KUKA KRL program: EPS_2_251806_MH45A_A_20260212042240.src

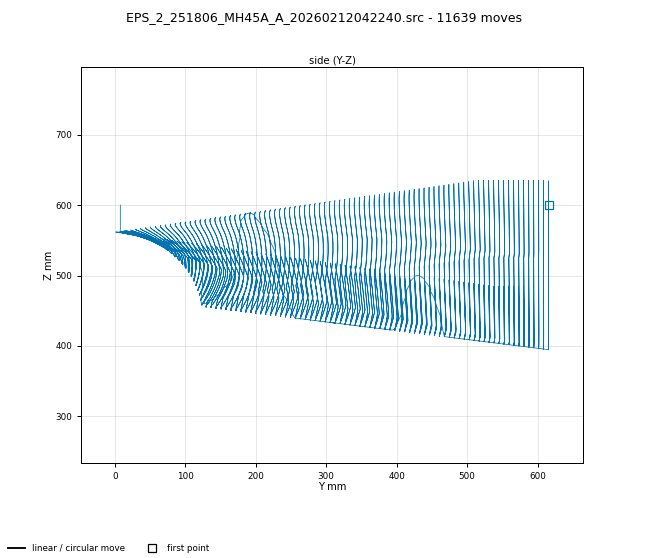
[picture p0: tool path of EPS_2_251806_MH45A_A_20260212042240.src, 11639 of 11641 moves have a stored position in this frame; points joined in program order, loops and branches not executed]
&ACCESS RVP
&REL 4
&COMMENT QRS 19112012
&PARAM EDITMASK = *
DEF PART()
EXT BAS (BAS_COMMAND :IN,REAL :IN )
INT I
BAS (#INITMOV,0 )

;KUKA QRS Post kuka4.cps  Date:22-06-2017 !

File_ID=3017

QRS_PRE_INIT()

;Init var - Until changes are made in qrs_pre_init
Outlet_Square_prg=0
Inlet_1_Square_prg=0
Inlet_2_Square_prg=0
Inlet_3_Square_prg=0
Inlet_4_Square_prg=0
Inlet_5_Square_prg=0

Outlet_1={X 0.000, Y 515.340, Z 534.500, B 0.000, E1 0.000 }
Inlet_1={X 0.000, Y 533.470, Z 284.500, B 0.000, E1 180.000 }
Outlet_1_type=201
Inlet_1_type=201
;QRS#1=Sidecore dimensions
;QRS#2=200-8" PVC SDR 35
;QRS#3=200-8" PVC SDR 35
;QRS#4=
;QRS#5=
;QRS#6=
;QRS#7=
;QRS#8=
;QRS#9=12-08 PSX
;QRS#10=12-08 PSX
;QRS#11=
;QRS#12=
;QRS#13=
;QRS#14=
;QRS#15=
;QRS#16=1220x127x914 3'
;QRS#17=EPS Height
;QRS#18=635
;QRS#19=*
;QRS#20= UPDATED VERSION 22-06-2017
;QRS#21=*
Outlet_Square=0100
Inlet_1_Square=0100
Inlet_2_Square=0
Inlet_3_Square=0
Inlet_4_Square=0
Inlet_5_Square=0
Mill_Square=1
Outlet_Square_Prg=204
Inlet_1_Square_prg=204

QRS_INIT()

$ADVANCE=5

; T1
PTP {E1 173.608,E2 173.608}
PTP {X 0,Y 615.507,A -85,B 0,C 180,E1 173.608,E2 173.608,E3 0,E4 0,E5 0,E6 0}
QRS_SPEED_INIT()
LIN {X 0,Y 615.507,Z 600,A -85,B 0,C 180,E1 173.608,E2 173.608,E3 0,E4 0,E5 0,E6 0} C_VEL
LIN {X 0,Y 615.507,Z 404.876,A -85,B 0,C 180,E1 173.608,E2 173.608} C_VEL
LIN {X 0,Y 615.507,Z 396.699,A -85,B 0,C 180,E1 173.608,E2 173.608} C_VEL
LIN {X 0,Y 615.491,Z 394.699,A -85,B 0,C 180,E1 173.422,E2 173.422} C_VEL
LIN {X 0,Y 615.482,Z 394.699,A -85,B 0,C 180,E1 170.801,E2 170.801} C_VEL
LIN {X 0,Y 615.49,Z 394.7,A -85,B 0,C 180,E1 168.139,E2 168.139} C_VEL
LIN {X 0,Y 615.496,Z 394.696,A -85,B 0,C 180,E1 165.451,E2 165.451} C_VEL
LIN {X 0,Y 615.497,Z 394.697,A -85,B 0,C 180,E1 162.73,E2 162.73} C_VEL
LIN {X 0,Y 615.486,Z 394.7,A -85,B 0,C 180,E1 159.967,E2 159.967} C_VEL
LIN {X 0,Y 615.477,Z 394.699,A -85,B 0,C 180,E1 157.155,E2 157.155} C_VEL
LIN {X 0,Y 615.496,Z 394.7,A -85,B 0,C 180,E1 154.43,E2 154.43} C_VEL
LIN {X 0,Y 615.497,Z 394.697,A -85,B 0,C 180,E1 151.549,E2 151.549} C_VEL
LIN {X 0,Y 615.491,Z 394.697,A -85,B 0,C 180,E1 148.914,E2 148.914} C_VEL
LIN {X 0,Y 615.485,Z 394.698,A -85,B 0,C 180,E1 146.467,E2 146.467} C_VEL
LIN {X 0,Y 615.49,Z 394.697,A -85,B 0,C 180,E1 143.575,E2 143.575} C_VEL
LIN {X 0,Y 615.481,Z 394.7,A -85,B 0,C 180,E1 140.939,E2 140.939} C_VEL
LIN {X 0,Y 615.495,Z 394.7,A -85,B 0,C 180,E1 138.527,E2 138.527} C_VEL
LIN {X 0,Y 615.494,Z 394.696,A -85,B 0,C 180,E1 135.851,E2 135.851} C_VEL
LIN {X 0,Y 615.487,Z 394.699,A -85,B 0,C 180,E1 133.047,E2 133.047} C_VEL
LIN {X 0,Y 615.479,Z 394.699,A -85,B 0,C 180,E1 130.607,E2 130.607} C_VEL
LIN {X 0,Y 615.488,Z 394.702,A -85,B 0,C 180,E1 128.012,E2 128.012} C_VEL
LIN {X 0,Y 615.486,Z 394.699,A -85,B 0,C 180,E1 125.616,E2 125.616} C_VEL
LIN {X 0,Y 615.479,Z 394.699,A -85,B 0,C 180,E1 123.237,E2 123.237} C_VEL
LIN {X 0,Y 615.493,Z 394.697,A -85,B 0,C 180,E1 120.92,E2 120.92} C_VEL
LIN {X 0,Y 615.497,Z 394.7,A -85,B 0,C 180,E1 118.451,E2 118.451} C_VEL
LIN {X 0,Y 615.492,Z 394.697,A -85,B 0,C 180,E1 115.569,E2 115.569} C_VEL
LIN {X 0,Y 615.49,Z 394.697,A -85,B 0,C 180,E1 112.845,E2 112.845} C_VEL
LIN {X 0,Y 615.487,Z 394.702,A -85,B 0,C 180,E1 110.033,E2 110.033} C_VEL
LIN {X 0,Y 615.477,Z 394.699,A -85,B 0,C 180,E1 107.271,E2 107.271} C_VEL
LIN {X 0,Y 615.49,Z 394.7,A -85,B 0,C 180,E1 104.549,E2 104.549} C_VEL
LIN {X 0,Y 615.494,Z 394.696,A -85,B 0,C 180,E1 101.861,E2 101.861} C_VEL
LIN {X 0,Y 615.487,Z 394.736,A -85,B 0,C 180,E1 101.235,E2 101.235} C_VEL
LIN {X 0,Y 615.485,Z 406.659,A -85,B 0,C 180,E1 100.84,E2 100.84} C_VEL
LIN {X 0,Y 615.494,Z 419.193,A -85,B 0,C 180,E1 100.277,E2 100.277} C_VEL
LIN {X 0,Y 615.493,Z 430.575,A -85,B 0,C 180,E1 99.613,E2 99.613} C_VEL
LIN {X 0,Y 615.498,Z 440.821,A -85,B 0,C 180,E1 98.867,E2 98.867} C_VEL
LIN {X 0,Y 615.499,Z 450.033,A -85,B 0,C 180,E1 98.041,E2 98.041} C_VEL
LIN {X 0,Y 615.499,Z 458.891,A -85,B 0,C 180,E1 97.057,E2 97.057} C_VEL
LIN {X 0,Y 615.497,Z 466.123,A -85,B 0,C 180,E1 96.063,E2 96.063} C_VEL
LIN {X 0,Y 615.497,Z 470.957,A -85,B 0,C 180,E1 95.241,E2 95.241} C_VEL
LIN {X 0,Y 615.494,Z 475.657,A -85,B 0,C 180,E1 94.256,E2 94.256} C_VEL
LIN {X 0,Y 615.494,Z 479.254,A -85,B 0,C 180,E1 93.273,E2 93.273} C_VEL
LIN {X 0,Y 615.496,Z 481.115,A -85,B 0,C 180,E1 92.618,E2 92.618} C_VEL
LIN {X 0,Y 615.499,Z 482.533,A -85,B 0,C 180,E1 91.963,E2 91.963} C_VEL
LIN {X 0,Y 615.496,Z 484.141,A -85,B 0,C 180,E1 90.654,E2 90.654} C_VEL
LIN {X 0,Y 615.495,Z 484.384,A -85,B 0,C 180,E1 90,E2 90} C_VEL
LIN {X 0,Y 615.495,Z 484.206,A -85,B 0,C 180,E1 89.346,E2 89.346} C_VEL
LIN {X 0,Y 615.499,Z 482.682,A -85,B 0,C 180,E1 88.037,E2 88.037} C_VEL
LIN {X 0,Y 615.498,Z 481.341,A -85,B 0,C 180,E1 87.382,E2 87.382} C_VEL
LIN {X 0,Y 615.496,Z 478.494,A -85,B 0,C 180,E1 86.399,E2 86.399} C_VEL
LIN {X 0,Y 615.499,Z 474.634,A -85,B 0,C 180,E1 85.416,E2 85.416} C_VEL
LIN {X 0,Y 615.498,Z 469.652,A -85,B 0,C 180,E1 84.43,E2 84.43} C_VEL
LIN {X 0,Y 615.496,Z 463.208,A -85,B 0,C 180,E1 83.418,E2 83.418} C_VEL
LIN {X 0,Y 615.497,Z 455.537,A -85,B 0,C 180,E1 82.455,E2 82.455} C_VEL
LIN {X 0,Y 615.498,Z 445.759,A -85,B 0,C 180,E1 81.464,E2 81.464} C_VEL
LIN {X 0,Y 615.498,Z 435.493,A -85,B 0,C 180,E1 80.636,E2 80.636} C_VEL
LIN {X 0,Y 615.492,Z 423.93,A -85,B 0,C 180,E1 79.889,E2 79.889} C_VEL
LIN {X 0,Y 615.485,Z 412.104,A -85,B 0,C 180,E1 79.294,E2 79.294} C_VEL
LIN {X 0,Y 615.486,Z 399.16,A -85,B 0,C 180,E1 78.807,E2 78.807} C_VEL
LIN {X 0,Y 615.485,Z 394.699,A -85,B 0,C 180,E1 78.661,E2 78.661} C_VEL
LIN {X 0,Y 615.499,Z 394.696,A -85,B 0,C 180,E1 76.064,E2 76.064} C_VEL
LIN {X 0,Y 615.481,Z 394.699,A -85,B 0,C 180,E1 73.413,E2 73.413} C_VEL
LIN {X 0,Y 615.483,Z 394.699,A -85,B 0,C 180,E1 70.662,E2 70.662} C_VEL
LIN {X 0,Y 615.495,Z 394.7,A -85,B 0,C 180,E1 67.864,E2 67.864} C_VEL
LIN {X 0,Y 615.489,Z 394.697,A -85,B 0,C 180,E1 65.008,E2 65.008} C_VEL
LIN {X 0,Y 615.488,Z 394.698,A -85,B 0,C 180,E1 62.823,E2 62.823} C_VEL
LIN {X 0,Y 615.499,Z 394.697,A -85,B 0,C 180,E1 60.204,E2 60.204} C_VEL
LIN {X 0,Y 615.481,Z 394.699,A -85,B 0,C 180,E1 57.542,E2 57.542} C_VEL
LIN {X 0,Y 615.499,Z 394.699,A -85,B 0,C 180,E1 55.186,E2 55.186} C_VEL
LIN {X 0,Y 615.488,Z 394.699,A -85,B 0,C 180,E1 52.758,E2 52.758} C_VEL
LIN {X 0,Y 615.497,Z 394.699,A -85,B 0,C 180,E1 49.91,E2 49.91} C_VEL
LIN {X 0,Y 615.496,Z 394.7,A -85,B 0,C 180,E1 47.648,E2 47.648} C_VEL
LIN {X 0,Y 615.481,Z 394.699,A -85,B 0,C 180,E1 44.931,E2 44.931} C_VEL
LIN {X 0,Y 615.487,Z 394.698,A -85,B 0,C 180,E1 42.08,E2 42.08} C_VEL
LIN {X 0,Y 615.477,Z 394.699,A -85,B 0,C 180,E1 39.751,E2 39.751} C_VEL
LIN {X 0,Y 615.486,Z 394.7,A -85,B 0,C 180,E1 36.936,E2 36.936} C_VEL
LIN {X 0,Y 615.494,Z 394.7,A -85,B 0,C 180,E1 34.022,E2 34.022} C_VEL
LIN {X 0,Y 615.489,Z 394.7,A -85,B 0,C 180,E1 31.686,E2 31.686} C_VEL
LIN {X 0,Y 615.492,Z 394.697,A -85,B 0,C 180,E1 29.406,E2 29.406} C_VEL
LIN {X 0,Y 615.495,Z 394.7,A -85,B 0,C 180,E1 26.444,E2 26.444} C_VEL
LIN {X 0,Y 615.486,Z 394.699,A -85,B 0,C 180,E1 23.557,E2 23.557} C_VEL
LIN {X 0,Y 615.484,Z 394.698,A -85,B 0,C 180,E1 20.731,E2 20.731} C_VEL
LIN {X 0,Y 615.49,Z 394.701,A -85,B 0,C 180,E1 17.957,E2 17.957} C_VEL
LIN {X 0,Y 615.486,Z 394.698,A -85,B 0,C 180,E1 15.226,E2 15.226} C_VEL
LIN {X 0,Y 615.494,Z 394.698,A -85,B 0,C 180,E1 12.53,E2 12.53} C_VEL
LIN {X 0,Y 615.481,Z 394.7,A -85,B 0,C 180,E1 9.862,E2 9.862} C_VEL
LIN {X 0,Y 615.484,Z 394.7,A -85,B 0,C 180,E1 7.216,E2 7.216} C_VEL
LIN {X 0,Y 615.489,Z 394.697,A -85,B 0,C 180,E1 4.585,E2 4.585} C_VEL
LIN {X 0,Y 615.484,Z 394.7,A -85,B 0,C 180,E1 1.963,E2 1.963} C_VEL
LIN {X 0,Y 615.485,Z 394.698,A -85,B 0,C 180,E1 -0.654,E2 -0.654} C_VEL
LIN {X 0,Y 615.498,Z 394.698,A -85,B 0,C 180,E1 -3.273,E2 -3.273} C_VEL
LIN {X 0,Y 615.483,Z 394.698,A -85,B 0,C 180,E1 -5.899,E2 -5.899} C_VEL
LIN {X 0,Y 615.486,Z 394.701,A -85,B 0,C 180,E1 -8.537,E2 -8.537} C_VEL
LIN {X 0,Y 615.486,Z 394.698,A -85,B 0,C 180,E1 -11.193,E2 -11.193} C_VEL
LIN {X 0,Y 615.487,Z 394.699,A -85,B 0,C 180,E1 -13.932,E2 -13.932} C_VEL
LIN {X 0,Y 615.487,Z 394.698,A -85,B 0,C 180,E1 -16.587,E2 -16.587} C_VEL
LIN {X 0,Y 615.493,Z 394.697,A -85,B 0,C 180,E1 -19.338,E2 -19.338} C_VEL
LIN {X 0,Y 615.494,Z 394.699,A -85,B 0,C 180,E1 -22.347,E2 -22.347} C_VEL
LIN {X 0,Y 615.477,Z 394.7,A -85,B 0,C 180,E1 -24.992,E2 -24.992} C_VEL
LIN {X 0,Y 615.485,Z 394.698,A -85,B 0,C 180,E1 -27.177,E2 -27.177} C_VEL
LIN {X 0,Y 615.481,Z 394.701,A -85,B 0,C 180,E1 -29.793,E2 -29.793} C_VEL
LIN {X 0,Y 615.487,Z 394.698,A -85,B 0,C 180,E1 -32.458,E2 -32.458} C_VEL
LIN {X 0,Y 615.49,Z 394.7,A -85,B 0,C 180,E1 -34.815,E2 -34.815} C_VEL
LIN {X 0,Y 615.493,Z 394.698,A -85,B 0,C 180,E1 -37.242,E2 -37.242} C_VEL
LIN {X 0,Y 615.491,Z 394.7,A -85,B 0,C 180,E1 -40.089,E2 -40.089} C_VEL
LIN {X 0,Y 615.498,Z 394.7,A -85,B 0,C 180,E1 -42.352,E2 -42.352} C_VEL
LIN {X 0,Y 615.485,Z 394.698,A -85,B 0,C 180,E1 -45.069,E2 -45.069} C_VEL
LIN {X 0,Y 615.481,Z 394.7,A -85,B 0,C 180,E1 -47.921,E2 -47.921} C_VEL
LIN {X 0,Y 615.494,Z 394.695,A -85,B 0,C 180,E1 -50.25,E2 -50.25} C_VEL
LIN {X 0,Y 615.495,Z 394.699,A -85,B 0,C 180,E1 -53.063,E2 -53.063} C_VEL
LIN {X 0,Y 615.481,Z 394.823,A -85,B 0,C 180,E1 -54.534,E2 -54.534} C_VEL
LIN {X 0,Y 615.489,Z 408.627,A -85,B 0,C 180,E1 -57.154,E2 -57.154} C_VEL
LIN {X 0,Y 615.476,Z 422.322,A -85,B 0,C 180,E1 -59.839,E2 -59.839} C_VEL
LIN {X 0,Y 615.481,Z 436.017,A -85,B 0,C 180,E1 -62.454,E2 -62.454} C_VEL
LIN {X 0,Y 615.497,Z 449.706,A -85,B 0,C 180,E1 -65.009,E2 -65.009} C_VEL
LIN {X 0,Y 615.487,Z 465.338,A -85,B 0,C 180,E1 -67.864,E2 -67.864} C_VEL
LIN {X 0,Y 615.492,Z 480.954,A -85,B 0,C 180,E1 -70.662,E2 -70.662} C_VEL
LIN {X 0,Y 615.492,Z 496.556,A -85,B 0,C 180,E1 -73.413,E2 -73.413} C_VEL
LIN {X 0,Y 615.498,Z 512.142,A -85,B 0,C 180,E1 -76.126,E2 -76.126} C_VEL
LIN {X 0,Y 615.482,Z 524.941,A -85,B 0,C 180,E1 -78.327,E2 -78.327} C_VEL
LIN {X 0,Y 615.477,Z 538.242,A -85,B 0,C 180,E1 -78.557,E2 -78.557} C_VEL
LIN {X 0,Y 615.489,Z 551.335,A -85,B 0,C 180,E1 -78.922,E2 -78.922} C_VEL
LIN {X 0,Y 615.48,Z 563.13,A -85,B 0,C 180,E1 -79.383,E2 -79.383} C_VEL
LIN {X 0,Y 615.486,Z 574.575,A -85,B 0,C 180,E1 -79.972,E2 -79.972} C_VEL
LIN {X 0,Y 615.499,Z 586.021,A -85,B 0,C 180,E1 -80.719,E2 -80.719} C_VEL
LIN {X 0,Y 615.498,Z 595.257,A -85,B 0,C 180,E1 -81.464,E2 -81.464} C_VEL
LIN {X 0,Y 615.499,Z 603.654,A -85,B 0,C 180,E1 -82.29,E2 -82.29} C_VEL
LIN {X 0,Y 615.497,Z 611.69,A -85,B 0,C 180,E1 -83.259,E2 -83.259} C_VEL
LIN {X 0,Y 615.498,Z 617.423,A -85,B 0,C 180,E1 -84.102,E2 -84.102} C_VEL
LIN {X 0,Y 615.497,Z 622.872,A -85,B 0,C 180,E1 -85.087,E2 -85.087} C_VEL
LIN {X 0,Y 615.496,Z 627.141,A -85,B 0,C 180,E1 -86.072,E2 -86.072} C_VEL
LIN {X 0,Y 615.495,Z 629.399,A -85,B 0,C 180,E1 -86.727,E2 -86.727} C_VEL
LIN {X 0,Y 615.497,Z 631.233,A -85,B 0,C 180,E1 -87.382,E2 -87.382} C_VEL
LIN {X 0,Y 615.497,Z 632.608,A -85,B 0,C 180,E1 -88.037,E2 -88.037} C_VEL
LIN {X 0,Y 615.496,Z 634.174,A -85,B 0,C 180,E1 -89.346,E2 -89.346} C_VEL
LIN {X 0,Y 615.494,Z 634.389,A -85,B 0,C 180,E1 -90,E2 -90} C_VEL
LIN {X 0,Y 615.496,Z 633.58,A -85,B 0,C 180,E1 -91.309,E2 -91.309} C_VEL
LIN {X 0,Y 615.497,Z 632.608,A -85,B 0,C 180,E1 -91.963,E2 -91.963} C_VEL
LIN {X 0,Y 615.497,Z 631.233,A -85,B 0,C 180,E1 -92.618,E2 -92.618} C_VEL
LIN {X 0,Y 615.496,Z 628.349,A -85,B 0,C 180,E1 -93.601,E2 -93.601} C_VEL
LIN {X 0,Y 615.498,Z 624.441,A -85,B 0,C 180,E1 -94.585,E2 -94.585} C_VEL
LIN {X 0,Y 615.499,Z 619.404,A -85,B 0,C 180,E1 -95.57,E2 -95.57} C_VEL
LIN {X 0,Y 615.497,Z 612.869,A -85,B 0,C 180,E1 -96.583,E2 -96.583} C_VEL
LIN {X 0,Y 615.497,Z 605.132,A -85,B 0,C 180,E1 -97.545,E2 -97.545} C_VEL
LIN {X 0,Y 615.498,Z 597.044,A -85,B 0,C 180,E1 -98.371,E2 -98.371} C_VEL
LIN {X 0,Y 615.499,Z 587.166,A -85,B 0,C 180,E1 -99.199,E2 -99.199} C_VEL
LIN {X 0,Y 615.488,Z 575.98,A -85,B 0,C 180,E1 -99.945,E2 -99.945} C_VEL
LIN {X 0,Y 615.478,Z 565.022,A -85,B 0,C 180,E1 -100.527,E2 -100.527} C_VEL
LIN {X 0,Y 615.489,Z 552.502,A -85,B 0,C 180,E1 -101.04,E2 -101.04} C_VEL
LIN {X 0,Y 615.477,Z 540.062,A -85,B 0,C 180,E1 -101.402,E2 -101.402} C_VEL
LIN {X 0,Y 615.481,Z 526.459,A -85,B 0,C 180,E1 -101.652,E2 -101.652} C_VEL
LIN {X 0,Y 615.483,Z 524.798,A -85,B 0,C 180,E1 -101.694,E2 -101.694} C_VEL
LIN {X 0,Y 615.48,Z 510.016,A -85,B 0,C 180,E1 -104.243,E2 -104.243} C_VEL
LIN {X 0,Y 615.494,Z 494.604,A -85,B 0,C 180,E1 -106.928,E2 -106.928} C_VEL
LIN {X 0,Y 615.495,Z 479.001,A -85,B 0,C 180,E1 -109.685,E2 -109.685} C_VEL
LIN {X 0,Y 615.494,Z 462.801,A -85,B 0,C 180,E1 -112.595,E2 -112.595} C_VEL
LIN {X 0,Y 615.485,Z 448.151,A -85,B 0,C 180,E1 -115.279,E2 -115.279} C_VEL
LIN {X 0,Y 615.493,Z 434.06,A -85,B 0,C 180,E1 -117.915,E2 -117.915} C_VEL
LIN {X 0,Y 615.478,Z 420.365,A -85,B 0,C 180,E1 -120.54,E2 -120.54} C_VEL
LIN {X 0,Y 615.491,Z 406.663,A -85,B 0,C 180,E1 -123.236,E2 -123.236} C_VEL
LIN {X 0,Y 615.482,Z 394.698,A -85,B 0,C 180,E1 -125.516,E2 -125.516} C_VEL
LIN {X 0,Y 615.498,Z 394.699,A -85,B 0,C 180,E1 -128.068,E2 -128.068} C_VEL
LIN {X 0,Y 615.491,Z 394.697,A -85,B 0,C 180,E1 -130.606,E2 -130.606} C_VEL
LIN {X 0,Y 615.491,Z 394.698,A -85,B 0,C 180,E1 -133.245,E2 -133.245} C_VEL
LIN {X 0,Y 615.484,Z 394.698,A -85,B 0,C 180,E1 -136.003,E2 -136.003} C_VEL
LIN {X 0,Y 615.485,Z 394.7,A -85,B 0,C 180,E1 -138.526,E2 -138.526} C_VEL
LIN {X 0,Y 615.484,Z 394.7,A -85,B 0,C 180,E1 -141.095,E2 -141.095} C_VEL
LIN {X 0,Y 615.489,Z 394.697,A -85,B 0,C 180,E1 -143.575,E2 -143.575} C_VEL
LIN {X 0,Y 615.494,Z 394.697,A -85,B 0,C 180,E1 -146.465,E2 -146.465} C_VEL
LIN {X 0,Y 615.49,Z 394.698,A -85,B 0,C 180,E1 -149.08,E2 -149.08} C_VEL
LIN {X 0,Y 615.498,Z 394.699,A -85,B 0,C 180,E1 -151.549,E2 -151.549} C_VEL
LIN {X 0,Y 615.484,Z 394.7,A -85,B 0,C 180,E1 -154.433,E2 -154.433} C_VEL
LIN {X 0,Y 615.48,Z 394.699,A -85,B 0,C 180,E1 -157.155,E2 -157.155} C_VEL
LIN {X 0,Y 615.491,Z 394.701,A -85,B 0,C 180,E1 -159.967,E2 -159.967} C_VEL
LIN {X 0,Y 615.495,Z 394.696,A -85,B 0,C 180,E1 -162.73,E2 -162.73} C_VEL
LIN {X 0,Y 615.497,Z 394.697,A -85,B 0,C 180,E1 -165.451,E2 -165.451} C_VEL
LIN {X 0,Y 615.484,Z 394.699,A -85,B 0,C 180,E1 -168.139,E2 -168.139} C_VEL
LIN {X 0,Y 615.479,Z 394.7,A -85,B 0,C 180,E1 -170.801,E2 -170.801} C_VEL
LIN {X 0,Y 615.492,Z 394.697,A -85,B 0,C 180,E1 -173.443,E2 -173.443} C_VEL
LIN {X 0,Y 615.49,Z 394.698,A -85,B 0,C 180,E1 -176.072,E2 -176.072} C_VEL
LIN {X 0,Y 615.495,Z 394.696,A -85,B 0,C 180,E1 -178.691,E2 -178.691} C_VEL
LIN {X 0,Y 615.496,Z 394.698,A -85,B 0,C 180,E1 -181.309,E2 -181.309} C_VEL
LIN {X 0,Y 615.48,Z 394.699,A -85,B 0,C 180,E1 -183.929,E2 -183.929} C_VEL
LIN {X 0,Y 615.491,Z 394.699,A -85,B 0,C 180,E1 -186.578,E2 -186.578} C_VEL
LIN {X 0,Y 614.81,Z 394.846,A -85,B 0,C 180,E1 -187.124,E2 -187.124} C_VEL
LIN {X 0,Y 611.97,Z 395.257,A -85,B 0,C 180,E1 -188.01,E2 -188.01} C_VEL
LIN {X 0,Y 609.579,Z 395.567,A -85,B 0,C 180,E1 -188.722,E2 -188.722} C_VEL
LIN {X 0,Y 608.546,Z 395.685,A -85,B 0,C 180,E1 -189.272,E2 -189.272} C_VEL
LIN {X 0,Y 608.458,Z 395.694,A -85,B 0,C 180,E1 -189.458,E2 -189.458} C_VEL
LIN {X 0,Y 608.467,Z 395.694,A -85,B 0,C 180,E1 -192,E2 -192} C_VEL
LIN {X 0,Y 608.482,Z 395.693,A -85,B 0,C 180,E1 -194.72,E2 -194.72} C_VEL
LIN {X 0,Y 608.459,Z 395.695,A -85,B 0,C 180,E1 -197.476,E2 -197.476} C_VEL
LIN {X 0,Y 608.464,Z 395.696,A -85,B 0,C 180,E1 -200.274,E2 -200.274} C_VEL
LIN {X 0,Y 608.463,Z 395.696,A -85,B 0,C 180,E1 -202.476,E2 -202.476} C_VEL
LIN {X 0,Y 608.451,Z 395.697,A -85,B 0,C 180,E1 -205.301,E2 -205.301} C_VEL
LIN {X 0,Y 608.451,Z 395.697,A -85,B 0,C 180,E1 -207.518,E2 -207.518} C_VEL
LIN {X 0,Y 608.475,Z 395.693,A -85,B 0,C 180,E1 -209.972,E2 -209.972} C_VEL
LIN {X 0,Y 608.468,Z 395.693,A -85,B 0,C 180,E1 -212.523,E2 -212.523} C_VEL
LIN {X 0,Y 608.441,Z 395.698,A -85,B 0,C 180,E1 -215.278,E2 -215.278} C_VEL
LIN {X 0,Y 608.472,Z 395.693,A -85,B 0,C 180,E1 -217.746,E2 -217.746} C_VEL
LIN {X 0,Y 608.449,Z 395.699,A -85,B 0,C 180,E1 -220.328,E2 -220.328} C_VEL
LIN {X 0,Y 608.485,Z 395.692,A -85,B 0,C 180,E1 -223.31,E2 -223.31} C_VEL
LIN {X 0,Y 608.477,Z 395.692,A -85,B 0,C 180,E1 -226.131,E2 -226.131} C_VEL
LIN {X 0,Y 608.458,Z 395.698,A -85,B 0,C 180,E1 -228.823,E2 -228.823} C_VEL
LIN {X 0,Y 608.476,Z 395.692,A -85,B 0,C 180,E1 -231.412,E2 -231.412} C_VEL
LIN {X 0,Y 608.452,Z 395.697,A -85,B 0,C 180,E1 -233.954,E2 -233.954} C_VEL
LIN {X 0,Y 608.451,Z 395.698,A -85,B 0,C 180,E1 -236.328,E2 -236.328} C_VEL
LIN {X 0,Y 608.45,Z 395.696,A -85,B 0,C 180,E1 -238.732,E2 -238.732} C_VEL
LIN {X 0,Y 608.482,Z 395.693,A -85,B 0,C 180,E1 -241.379,E2 -241.379} C_VEL
LIN {X 0,Y 608.478,Z 395.692,A -85,B 0,C 180,E1 -244.278,E2 -244.278} C_VEL
LIN {X 0,Y 608.454,Z 395.698,A -85,B 0,C 180,E1 -246.876,E2 -246.876} C_VEL
LIN {X 0,Y 608.466,Z 395.694,A -85,B 0,C 180,E1 -249.323,E2 -249.323} C_VEL
LIN {X 0,Y 608.453,Z 395.696,A -85,B 0,C 180,E1 -251.828,E2 -251.828} C_VEL
LIN {X 0,Y 608.469,Z 395.694,A -85,B 0,C 180,E1 -254.594,E2 -254.594} C_VEL
LIN {X 0,Y 608.48,Z 395.694,A -85,B 0,C 180,E1 -257.323,E2 -257.323} C_VEL
LIN {X 0,Y 608.464,Z 395.695,A -85,B 0,C 180,E1 -258.655,E2 -258.655} C_VEL
LIN {X 0,Y 608.519,Z 407.477,A -85,B 0,C 180,E1 -259.059,E2 -259.059} C_VEL
LIN {X 0,Y 608.506,Z 419.367,A -85,B 0,C 180,E1 -259.603,E2 -259.603} C_VEL
LIN {X 0,Y 608.506,Z 430.787,A -85,B 0,C 180,E1 -260.275,E2 -260.275} C_VEL
LIN {X 0,Y 608.474,Z 441.083,A -85,B 0,C 180,E1 -261.029,E2 -261.029} C_VEL
LIN {X 0,Y 608.464,Z 450.35,A -85,B 0,C 180,E1 -261.866,E2 -261.866} C_VEL
LIN {X 0,Y 608.466,Z 459.323,A -85,B 0,C 180,E1 -262.867,E2 -262.867} C_VEL
LIN {X 0,Y 608.444,Z 466.556,A -85,B 0,C 180,E1 -263.866,E2 -263.866} C_VEL
LIN {X 0,Y 608.462,Z 471.435,A -85,B 0,C 180,E1 -264.698,E2 -264.698} C_VEL
LIN {X 0,Y 608.439,Z 476.179,A -85,B 0,C 180,E1 -265.694,E2 -265.694} C_VEL
LIN {X 0,Y 608.425,Z 479.812,A -85,B 0,C 180,E1 -266.689,E2 -266.689} C_VEL
LIN {X 0,Y 608.425,Z 481.691,A -85,B 0,C 180,E1 -267.352,E2 -267.352} C_VEL
LIN {X 0,Y 608.444,Z 483.127,A -85,B 0,C 180,E1 -268.014,E2 -268.014} C_VEL
LIN {X 0,Y 608.439,Z 484.752,A -85,B 0,C 180,E1 -269.338,E2 -269.338} C_VEL
LIN {X 0,Y 608.435,Z 484.995,A -85,B 0,C 180,E1 -270,E2 -270} C_VEL
LIN {X 0,Y 608.438,Z 484.815,A -85,B 0,C 180,E1 -270.662,E2 -270.662} C_VEL
LIN {X 0,Y 608.444,Z 483.276,A -85,B 0,C 180,E1 -271.986,E2 -271.986} C_VEL
LIN {X 0,Y 608.426,Z 481.919,A -85,B 0,C 180,E1 -272.648,E2 -272.648} C_VEL
LIN {X 0,Y 608.449,Z 479.042,A -85,B 0,C 180,E1 -273.642,E2 -273.642} C_VEL
LIN {X 0,Y 608.433,Z 475.144,A -85,B 0,C 180,E1 -274.638,E2 -274.638} C_VEL
LIN {X 0,Y 608.45,Z 470.113,A -85,B 0,C 180,E1 -275.634,E2 -275.634} C_VEL
LIN {X 0,Y 608.441,Z 463.794,A -85,B 0,C 180,E1 -276.633,E2 -276.633} C_VEL
LIN {X 0,Y 608.475,Z 455.879,A -85,B 0,C 180,E1 -277.633,E2 -277.633} C_VEL
LIN {X 0,Y 608.472,Z 446.036,A -85,B 0,C 180,E1 -278.636,E2 -278.636} C_VEL
LIN {X 0,Y 608.481,Z 435.714,A -85,B 0,C 180,E1 -279.473,E2 -279.473} C_VEL
LIN {X 0,Y 608.489,Z 424.099,A -85,B 0,C 180,E1 -280.229,E2 -280.229} C_VEL
LIN {X 0,Y 608.506,Z 412.237,A -85,B 0,C 180,E1 -280.83,E2 -280.83} C_VEL
LIN {X 0,Y 608.525,Z 399.267,A -85,B 0,C 180,E1 -281.323,E2 -281.323} C_VEL
LIN {X 0,Y 608.47,Z 395.695,A -85,B 0,C 180,E1 -281.45,E2 -281.45} C_VEL
LIN {X 0,Y 608.474,Z 395.693,A -85,B 0,C 180,E1 -284.037,E2 -284.037} C_VEL
LIN {X 0,Y 608.443,Z 395.699,A -85,B 0,C 180,E1 -286.784,E2 -286.784} C_VEL
LIN {X 0,Y 608.452,Z 395.695,A -85,B 0,C 180,E1 -289.571,E2 -289.571} C_VEL
LIN {X 0,Y 608.463,Z 395.695,A -85,B 0,C 180,E1 -292.476,E2 -292.476} C_VEL
LIN {X 0,Y 608.458,Z 395.695,A -85,B 0,C 180,E1 -294.571,E2 -294.571} C_VEL
LIN {X 0,Y 608.482,Z 395.692,A -85,B 0,C 180,E1 -297.207,E2 -297.207} C_VEL
LIN {X 0,Y 608.474,Z 395.693,A -85,B 0,C 180,E1 -299.972,E2 -299.972} C_VEL
LIN {X 0,Y 608.453,Z 395.697,A -85,B 0,C 180,E1 -302.88,E2 -302.88} C_VEL
LIN {X 0,Y 608.448,Z 395.696,A -85,B 0,C 180,E1 -305.277,E2 -305.277} C_VEL
LIN {X 0,Y 608.475,Z 395.693,A -85,B 0,C 180,E1 -307.746,E2 -307.746} C_VEL
LIN {X 0,Y 608.453,Z 395.697,A -85,B 0,C 180,E1 -310.329,E2 -310.329} C_VEL
LIN {X 0,Y 608.454,Z 395.695,A -85,B 0,C 180,E1 -312.96,E2 -312.96} C_VEL
LIN {X 0,Y 608.461,Z 395.695,A -85,B 0,C 180,E1 -315.736,E2 -315.736} C_VEL
LIN {X 0,Y 608.462,Z 395.697,A -85,B 0,C 180,E1 -318.658,E2 -318.658} C_VEL
LIN {X 0,Y 608.471,Z 395.695,A -85,B 0,C 180,E1 -321.76,E2 -321.76} C_VEL
LIN {X 0,Y 608.45,Z 395.699,A -85,B 0,C 180,E1 -323.954,E2 -323.954} C_VEL
LIN {X 0,Y 608.467,Z 395.694,A -85,B 0,C 180,E1 -326.329,E2 -326.329} C_VEL
LIN {X 0,Y 608.465,Z 395.694,A -85,B 0,C 180,E1 -328.73,E2 -328.73} C_VEL
LIN {X 0,Y 608.478,Z 395.695,A -85,B 0,C 180,E1 -331.38,E2 -331.38} C_VEL
LIN {X 0,Y 608.47,Z 395.694,A -85,B 0,C 180,E1 -334.28,E2 -334.28} C_VEL
LIN {X 0,Y 608.446,Z 395.697,A -85,B 0,C 180,E1 -336.876,E2 -336.876} C_VEL
LIN {X 0,Y 608.47,Z 395.693,A -85,B 0,C 180,E1 -339.321,E2 -339.321} C_VEL
LIN {X 0,Y 608.452,Z 395.697,A -85,B 0,C 180,E1 -341.828,E2 -341.828} C_VEL
LIN {X 0,Y 608.472,Z 395.693,A -85,B 0,C 180,E1 -344.594,E2 -344.594} C_VEL
LIN {X 0,Y 608.481,Z 395.694,A -85,B 0,C 180,E1 -347.323,E2 -347.323} C_VEL
LIN {X 0,Y 608.454,Z 395.695,A -85,B 0,C 180,E1 -350.023,E2 -350.023} C_VEL
LIN {X 0,Y 608.463,Z 395.696,A -85,B 0,C 180,E1 -352.701,E2 -352.701} C_VEL
LIN {X 0,Y 608.458,Z 395.695,A -85,B 0,C 180,E1 -355.362,E2 -355.362} C_VEL
LIN {X 0,Y 608.454,Z 395.697,A -85,B 0,C 180,E1 -358.014,E2 -358.014} C_VEL
LIN {X 0,Y 608.48,Z 395.692,A -85,B 0,C 180,E1 -360.662,E2 -360.662} C_VEL
LIN {X 0,Y 608.49,Z 395.692,A -85,B 0,C 180,E1 -363.311,E2 -363.311} C_VEL
LIN {X 0,Y 608.458,Z 395.695,A -85,B 0,C 180,E1 -365.967,E2 -365.967} C_VEL
LIN {X 0,Y 608.456,Z 395.696,A -85,B 0,C 180,E1 -368.636,E2 -368.636} C_VEL
LIN {X 0,Y 608.477,Z 395.693,A -85,B 0,C 180,E1 -371.324,E2 -371.324} C_VEL
LIN {X 0,Y 608.473,Z 395.693,A -85,B 0,C 180,E1 -374.037,E2 -374.037} C_VEL
LIN {X 0,Y 608.479,Z 395.694,A -85,B 0,C 180,E1 -376.783,E2 -376.783} C_VEL
LIN {X 0,Y 608.459,Z 395.694,A -85,B 0,C 180,E1 -379.57,E2 -379.57} C_VEL
LIN {X 0,Y 608.462,Z 395.695,A -85,B 0,C 180,E1 -382.476,E2 -382.476} C_VEL
LIN {X 0,Y 608.452,Z 395.696,A -85,B 0,C 180,E1 -384.571,E2 -384.571} C_VEL
LIN {X 0,Y 608.478,Z 395.693,A -85,B 0,C 180,E1 -387.207,E2 -387.207} C_VEL
LIN {X 0,Y 608.463,Z 395.694,A -85,B 0,C 180,E1 -389.97,E2 -389.97} C_VEL
LIN {X 0,Y 608.463,Z 395.695,A -85,B 0,C 180,E1 -392.522,E2 -392.522} C_VEL
LIN {X 0,Y 608.446,Z 395.696,A -85,B 0,C 180,E1 -395.278,E2 -395.278} C_VEL
LIN {X 0,Y 608.474,Z 395.693,A -85,B 0,C 180,E1 -397.746,E2 -397.746} C_VEL
LIN {X 0,Y 608.45,Z 395.697,A -85,B 0,C 180,E1 -400.329,E2 -400.329} C_VEL
LIN {X 0,Y 608.484,Z 395.694,A -85,B 0,C 180,E1 -403.31,E2 -403.31} C_VEL
LIN {X 0,Y 608.47,Z 395.693,A -85,B 0,C 180,E1 -406.13,E2 -406.13} C_VEL
LIN {X 0,Y 608.462,Z 395.696,A -85,B 0,C 180,E1 -408.824,E2 -408.824} C_VEL
LIN {X 0,Y 608.477,Z 395.692,A -85,B 0,C 180,E1 -411.412,E2 -411.412} C_VEL
LIN {X 0,Y 608.481,Z 395.693,A -85,B 0,C 180,E1 -414.318,E2 -414.318} C_VEL
LIN {X 0,Y 608.57,Z 402.886,A -85,B 0,C 180,E1 -415.737,E2 -415.737} C_VEL
LIN {X 0,Y 608.636,Z 416.452,A -85,B 0,C 180,E1 -418.305,E2 -418.305} C_VEL
LIN {X 0,Y 608.599,Z 430.147,A -85,B 0,C 180,E1 -420.987,E2 -420.987} C_VEL
LIN {X 0,Y 608.552,Z 443.842,A -85,B 0,C 180,E1 -423.601,E2 -423.601} C_VEL
LIN {X 0,Y 608.532,Z 457.537,A -85,B 0,C 180,E1 -426.158,E2 -426.158} C_VEL
LIN {X 0,Y 608.522,Z 471.232,A -85,B 0,C 180,E1 -428.666,E2 -428.666} C_VEL
LIN {X 0,Y 608.494,Z 485.749,A -85,B 0,C 180,E1 -431.278,E2 -431.278} C_VEL
LIN {X 0,Y 608.483,Z 500.579,A -85,B 0,C 180,E1 -433.907,E2 -433.907} C_VEL
LIN {X 0,Y 608.464,Z 516.23,A -85,B 0,C 180,E1 -436.644,E2 -436.644} C_VEL
LIN {X 0,Y 608.447,Z 525.156,A -85,B 0,C 180,E1 -438.19,E2 -438.19} C_VEL
LIN {X 0,Y 608.526,Z 538.353,A -85,B 0,C 180,E1 -438.424,E2 -438.424} C_VEL
LIN {X 0,Y 608.53,Z 550.913,A -85,B 0,C 180,E1 -438.776,E2 -438.776} C_VEL
LIN {X 0,Y 608.516,Z 561.952,A -85,B 0,C 180,E1 -439.203,E2 -439.203} C_VEL
LIN {X 0,Y 608.482,Z 573.328,A -85,B 0,C 180,E1 -439.771,E2 -439.771} C_VEL
LIN {X 0,Y 608.49,Z 583.93,A -85,B 0,C 180,E1 -440.443,E2 -440.443} C_VEL
LIN {X 0,Y 608.477,Z 593.598,A -85,B 0,C 180,E1 -441.197,E2 -441.197} C_VEL
LIN {X 0,Y 608.46,Z 602.414,A -85,B 0,C 180,E1 -442.033,E2 -442.033} C_VEL
LIN {X 0,Y 608.444,Z 610.998,A -85,B 0,C 180,E1 -443.034,E2 -443.034} C_VEL
LIN {X 0,Y 608.438,Z 617.866,A -85,B 0,C 180,E1 -444.033,E2 -444.033} C_VEL
LIN {X 0,Y 608.438,Z 623.365,A -85,B 0,C 180,E1 -445.03,E2 -445.03} C_VEL
LIN {X 0,Y 608.434,Z 627.676,A -85,B 0,C 180,E1 -446.026,E2 -446.026} C_VEL
LIN {X 0,Y 608.425,Z 629.956,A -85,B 0,C 180,E1 -446.689,E2 -446.689} C_VEL
LIN {X 0,Y 608.425,Z 631.809,A -85,B 0,C 180,E1 -447.352,E2 -447.352} C_VEL
LIN {X 0,Y 608.442,Z 633.201,A -85,B 0,C 180,E1 -448.014,E2 -448.014} C_VEL
LIN {X 0,Y 608.438,Z 634.784,A -85,B 0,C 180,E1 -449.338,E2 -449.338} C_VEL
LIN {X 0,Y 608.434,Z 635,A -85,B 0,C 180,E1 -450,E2 -450} C_VEL
LIN {X 0,Y 608.448,Z 634.184,A -85,B 0,C 180,E1 -451.324,E2 -451.324} C_VEL
LIN {X 0,Y 608.443,Z 633.201,A -85,B 0,C 180,E1 -451.986,E2 -451.986} C_VEL
LIN {X 0,Y 608.425,Z 631.809,A -85,B 0,C 180,E1 -452.648,E2 -452.648} C_VEL
LIN {X 0,Y 608.449,Z 628.896,A -85,B 0,C 180,E1 -453.642,E2 -453.642} C_VEL
LIN {X 0,Y 608.432,Z 624.95,A -85,B 0,C 180,E1 -454.638,E2 -454.638} C_VEL
LIN {X 0,Y 608.437,Z 618.876,A -85,B 0,C 180,E1 -455.801,E2 -455.801} C_VEL
LIN {X 0,Y 608.462,Z 612.234,A -85,B 0,C 180,E1 -456.799,E2 -456.799} C_VEL
LIN {X 0,Y 608.456,Z 603.988,A -85,B 0,C 180,E1 -457.8,E2 -457.8} C_VEL
LIN {X 0,Y 608.472,Z 595.535,A -85,B 0,C 180,E1 -458.636,E2 -458.636} C_VEL
LIN {X 0,Y 608.481,Z 585.089,A -85,B 0,C 180,E1 -459.473,E2 -459.473} C_VEL
LIN {X 0,Y 608.494,Z 574.754,A -85,B 0,C 180,E1 -460.145,E2 -460.145} C_VEL
LIN {X 0,Y 608.51,Z 563.271,A -85,B 0,C 180,E1 -460.74,E2 -460.74} C_VEL
LIN {X 0,Y 608.53,Z 550.909,A -85,B 0,C 180,E1 -461.224,E2 -461.224} C_VEL
LIN {X 0,Y 608.537,Z 537.434,A -85,B 0,C 180,E1 -461.597,E2 -461.597} C_VEL
LIN {X 0,Y 608.447,Z 525.156,A -85,B 0,C 180,E1 -461.81,E2 -461.81} C_VEL
LIN {X 0,Y 608.479,Z 508.404,A -85,B 0,C 180,E1 -464.721,E2 -464.721} C_VEL
LIN {X 0,Y 608.492,Z 492.753,A -85,B 0,C 180,E1 -467.476,E2 -467.476} C_VEL
LIN {X 0,Y 608.516,Z 479.057,A -85,B 0,C 180,E1 -469.92,E2 -469.92} C_VEL
LIN {X 0,Y 608.549,Z 463.408,A -85,B 0,C 180,E1 -472.761,E2 -472.761} C_VEL
LIN {X 0,Y 608.563,Z 447.351,A -85,B 0,C 180,E1 -475.738,E2 -475.738} C_VEL
LIN {X 0,Y 608.593,Z 432.081,A -85,B 0,C 180,E1 -478.64,E2 -478.64} C_VEL
LIN {X 0,Y 608.612,Z 418.408,A -85,B 0,C 180,E1 -481.308,E2 -481.308} C_VEL
LIN {X 0,Y 608.575,Z 409.237,A -85,B 0,C 180,E1 -483.07,E2 -483.07} C_VEL
LIN {X 0,Y 608.535,Z 396.068,A -85,B 0,C 180,E1 -485.576,E2 -485.576} C_VEL
LIN {X 0,Y 608.48,Z 395.693,A -85,B 0,C 180,E1 -485.682,E2 -485.682} C_VEL
LIN {X 0,Y 608.478,Z 395.692,A -85,B 0,C 180,E1 -488.588,E2 -488.588} C_VEL
LIN {X 0,Y 608.467,Z 395.696,A -85,B 0,C 180,E1 -491.342,E2 -491.342} C_VEL
LIN {X 0,Y 608.451,Z 395.696,A -85,B 0,C 180,E1 -494.263,E2 -494.263} C_VEL
LIN {X 0,Y 608.453,Z 395.695,A -85,B 0,C 180,E1 -497.04,E2 -497.04} C_VEL
LIN {X 0,Y 608.456,Z 395.697,A -85,B 0,C 180,E1 -499.697,E2 -499.697} C_VEL
LIN {X 0,Y 608.473,Z 395.693,A -85,B 0,C 180,E1 -502.254,E2 -502.254} C_VEL
LIN {X 0,Y 608.447,Z 395.696,A -85,B 0,C 180,E1 -504.722,E2 -504.722} C_VEL
LIN {X 0,Y 608.462,Z 395.695,A -85,B 0,C 180,E1 -507.478,E2 -507.478} C_VEL
LIN {X 0,Y 608.467,Z 395.695,A -85,B 0,C 180,E1 -510.22,E2 -510.22} C_VEL
LIN {X 0,Y 608.477,Z 395.693,A -85,B 0,C 180,E1 -512.794,E2 -512.794} C_VEL
LIN {X 0,Y 608.453,Z 395.696,A -85,B 0,C 180,E1 -515.429,E2 -515.429} C_VEL
LIN {X 0,Y 608.477,Z 395.692,A -85,B 0,C 180,E1 -518.309,E2 -518.309} C_VEL
LIN {X 0,Y 608.473,Z 395.693,A -85,B 0,C 180,E1 -521.284,E2 -521.284} C_VEL
LIN {X 0,Y 608.464,Z 395.695,A -85,B 0,C 180,E1 -523.906,E2 -523.906} C_VEL
LIN {X 0,Y 608.465,Z 395.694,A -85,B 0,C 180,E1 -526.644,E2 -526.644} C_VEL
LIN {X 0,Y 608.467,Z 395.695,A -85,B 0,C 180,E1 -529.35,E2 -529.35} C_VEL
LIN {X 0,Y 608.473,Z 395.693,A -85,B 0,C 180,E1 -532.033,E2 -532.033} C_VEL
LIN {X 0,Y 608.474,Z 395.695,A -85,B 0,C 180,E1 -534.698,E2 -534.698} C_VEL
LIN {X 0,Y 608.482,Z 395.692,A -85,B 0,C 180,E1 -537.352,E2 -537.352} C_VEL
LIN {X 0,Y 608.479,Z 395.694,A -85,B 0,C 180,E1 -540,E2 -540} C_VEL
LIN {X 0,Y 608.483,Z 395.691,A -85,B 0,C 180,E1 -542.648,E2 -542.648} C_VEL
LIN {X 0,Y 608.469,Z 395.696,A -85,B 0,C 180,E1 -545.302,E2 -545.302} C_VEL
LIN {X 0,Y 608.472,Z 395.693,A -85,B 0,C 180,E1 -547.967,E2 -547.967} C_VEL
LIN {X 0,Y 608.458,Z 395.694,A -85,B 0,C 180,E1 -549.458,E2 -549.458} C_VEL
LIN {X 0,Y 607.782,Z 395.779,A -85,B 0,C 180,E1 -550.011,E2 -550.011} C_VEL
LIN {X 0,Y 604.931,Z 396.135,A -85,B 0,C 180,E1 -550.907,E2 -550.907} C_VEL
LIN {X 0,Y 602.529,Z 396.435,A -85,B 0,C 180,E1 -551.629,E2 -551.629} C_VEL
LIN {X 0,Y 601.498,Z 396.561,A -85,B 0,C 180,E1 -552.186,E2 -552.186} C_VEL
LIN {X 0,Y 601.414,Z 396.572,A -85,B 0,C 180,E1 -552.374,E2 -552.374} C_VEL
LIN {X 0,Y 601.436,Z 396.572,A -85,B 0,C 180,E1 -554.897,E2 -554.897} C_VEL
LIN {X 0,Y 601.438,Z 396.572,A -85,B 0,C 180,E1 -556.986,E2 -556.986} C_VEL
LIN {X 0,Y 601.41,Z 396.573,A -85,B 0,C 180,E1 -559.809,E2 -559.809} C_VEL
LIN {X 0,Y 601.416,Z 396.572,A -85,B 0,C 180,E1 -562.683,E2 -562.683} C_VEL
LIN {X 0,Y 601.403,Z 396.573,A -85,B 0,C 180,E1 -564.879,E2 -564.879} C_VEL
LIN {X 0,Y 601.418,Z 396.572,A -85,B 0,C 180,E1 -567.362,E2 -567.362} C_VEL
LIN {X 0,Y 601.434,Z 396.569,A -85,B 0,C 180,E1 -570.164,E2 -570.164} C_VEL
LIN {X 0,Y 601.429,Z 396.571,A -85,B 0,C 180,E1 -572.716,E2 -572.716} C_VEL
LIN {X 0,Y 601.397,Z 396.577,A -85,B 0,C 180,E1 -575.112,E2 -575.112} C_VEL
LIN {X 0,Y 601.44,Z 396.57,A -85,B 0,C 180,E1 -577.419,E2 -577.419} C_VEL
LIN {X 0,Y 601.404,Z 396.574,A -85,B 0,C 180,E1 -579.996,E2 -579.996} C_VEL
LIN {X 0,Y 601.417,Z 396.573,A -85,B 0,C 180,E1 -582.67,E2 -582.67} C_VEL
LIN {X 0,Y 601.431,Z 396.572,A -85,B 0,C 180,E1 -585.482,E2 -585.482} C_VEL
LIN {X 0,Y 601.43,Z 396.57,A -85,B 0,C 180,E1 -588.407,E2 -588.407} C_VEL
LIN {X 0,Y 601.443,Z 396.571,A -85,B 0,C 180,E1 -590.876,E2 -590.876} C_VEL
LIN {X 0,Y 601.407,Z 396.573,A -85,B 0,C 180,E1 -593.417,E2 -593.417} C_VEL
LIN {X 0,Y 601.436,Z 396.57,A -85,B 0,C 180,E1 -596.064,E2 -596.064} C_VEL
LIN {X 0,Y 601.424,Z 396.572,A -85,B 0,C 180,E1 -598.545,E2 -598.545} C_VEL
LIN {X 0,Y 601.442,Z 396.57,A -85,B 0,C 180,E1 -601.373,E2 -601.373} C_VEL
LIN {X 0,Y 601.419,Z 396.571,A -85,B 0,C 180,E1 -604.132,E2 -604.132} C_VEL
LIN {X 0,Y 601.424,Z 396.572,A -85,B 0,C 180,E1 -606.59,E2 -606.59} C_VEL
LIN {X 0,Y 601.43,Z 396.57,A -85,B 0,C 180,E1 -609.478,E2 -609.478} C_VEL
LIN {X 0,Y 601.397,Z 396.576,A -85,B 0,C 180,E1 -612.312,E2 -612.312} C_VEL
LIN {X 0,Y 601.414,Z 396.574,A -85,B 0,C 180,E1 -614.409,E2 -614.409} C_VEL
LIN {X 0,Y 601.424,Z 396.572,A -85,B 0,C 180,E1 -617.172,E2 -617.172} C_VEL
LIN {X 0,Y 601.422,Z 396.574,A -85,B 0,C 180,E1 -618.542,E2 -618.542} C_VEL
LIN {X 0,Y 601.544,Z 408.71,A -85,B 0,C 180,E1 -618.981,E2 -618.981} C_VEL
LIN {X 0,Y 601.515,Z 420.946,A -85,B 0,C 180,E1 -619.566,E2 -619.566} C_VEL
LIN {X 0,Y 601.471,Z 432.073,A -85,B 0,C 180,E1 -620.245,E2 -620.245} C_VEL
LIN {X 0,Y 601.438,Z 441.091,A -85,B 0,C 180,E1 -620.923,E2 -620.923} C_VEL
LIN {X 0,Y 601.411,Z 450.356,A -85,B 0,C 180,E1 -621.77,E2 -621.77} C_VEL
LIN {X 0,Y 601.388,Z 459.33,A -85,B 0,C 180,E1 -622.783,E2 -622.783} C_VEL
LIN {X 0,Y 601.376,Z 466.471,A -85,B 0,C 180,E1 -623.78,E2 -623.78} C_VEL
LIN {X 0,Y 601.373,Z 471.44,A -85,B 0,C 180,E1 -624.635,E2 -624.635} C_VEL
LIN {X 0,Y 601.354,Z 476.183,A -85,B 0,C 180,E1 -625.643,E2 -625.643} C_VEL
LIN {X 0,Y 601.344,Z 479.816,A -85,B 0,C 180,E1 -626.65,E2 -626.65} C_VEL
LIN {X 0,Y 601.324,Z 481.693,A -85,B 0,C 180,E1 -627.32,E2 -627.32} C_VEL
LIN {X 0,Y 601.343,Z 483.128,A -85,B 0,C 180,E1 -627.991,E2 -627.991} C_VEL
LIN {X 0,Y 601.339,Z 484.753,A -85,B 0,C 180,E1 -629.33,E2 -629.33} C_VEL
LIN {X 0,Y 601.336,Z 484.996,A -85,B 0,C 180,E1 -630,E2 -630} C_VEL
LIN {X 0,Y 601.339,Z 484.815,A -85,B 0,C 180,E1 -630.67,E2 -630.67} C_VEL
LIN {X 0,Y 601.343,Z 483.276,A -85,B 0,C 180,E1 -632.009,E2 -632.009} C_VEL
LIN {X 0,Y 601.326,Z 481.917,A -85,B 0,C 180,E1 -632.68,E2 -632.68} C_VEL
LIN {X 0,Y 601.368,Z 479.043,A -85,B 0,C 180,E1 -633.685,E2 -633.685} C_VEL
LIN {X 0,Y 601.337,Z 475.144,A -85,B 0,C 180,E1 -634.693,E2 -634.693} C_VEL
LIN {X 0,Y 601.373,Z 470.113,A -85,B 0,C 180,E1 -635.701,E2 -635.701} C_VEL
LIN {X 0,Y 601.382,Z 463.789,A -85,B 0,C 180,E1 -636.711,E2 -636.711} C_VEL
LIN {X 0,Y 601.396,Z 455.877,A -85,B 0,C 180,E1 -637.723,E2 -637.723} C_VEL
LIN {X 0,Y 601.436,Z 446.029,A -85,B 0,C 180,E1 -638.738,E2 -638.738} C_VEL
LIN {X 0,Y 601.45,Z 435.708,A -85,B 0,C 180,E1 -639.585,E2 -639.585} C_VEL
LIN {X 0,Y 601.495,Z 424.091,A -85,B 0,C 180,E1 -640.349,E2 -640.349} C_VEL
LIN {X 0,Y 601.518,Z 412.229,A -85,B 0,C 180,E1 -640.958,E2 -640.958} C_VEL
LIN {X 0,Y 601.551,Z 399.258,A -85,B 0,C 180,E1 -641.456,E2 -641.456} C_VEL
LIN {X 0,Y 601.419,Z 396.575,A -85,B 0,C 180,E1 -641.544,E2 -641.544} C_VEL
LIN {X 0,Y 601.424,Z 396.57,A -85,B 0,C 180,E1 -644.205,E2 -644.205} C_VEL
LIN {X 0,Y 601.415,Z 396.574,A -85,B 0,C 180,E1 -646.986,E2 -646.986} C_VEL
LIN {X 0,Y 601.408,Z 396.574,A -85,B 0,C 180,E1 -649.809,E2 -649.809} C_VEL
LIN {X 0,Y 601.417,Z 396.572,A -85,B 0,C 180,E1 -652.683,E2 -652.683} C_VEL
LIN {X 0,Y 601.407,Z 396.573,A -85,B 0,C 180,E1 -654.878,E2 -654.878} C_VEL
LIN {X 0,Y 601.426,Z 396.571,A -85,B 0,C 180,E1 -657.867,E2 -657.867} C_VEL
LIN {X 0,Y 601.433,Z 396.569,A -85,B 0,C 180,E1 -660.164,E2 -660.164} C_VEL
LIN {X 0,Y 601.419,Z 396.574,A -85,B 0,C 180,E1 -662.714,E2 -662.714} C_VEL
LIN {X 0,Y 601.418,Z 396.573,A -85,B 0,C 180,E1 -665.115,E2 -665.115} C_VEL
LIN {X 0,Y 601.44,Z 396.569,A -85,B 0,C 180,E1 -667.419,E2 -667.419} C_VEL
LIN {X 0,Y 601.416,Z 396.573,A -85,B 0,C 180,E1 -669.995,E2 -669.995} C_VEL
LIN {X 0,Y 601.416,Z 396.572,A -85,B 0,C 180,E1 -672.67,E2 -672.67} C_VEL
LIN {X 0,Y 601.43,Z 396.573,A -85,B 0,C 180,E1 -675.482,E2 -675.482} C_VEL
LIN {X 0,Y 601.426,Z 396.571,A -85,B 0,C 180,E1 -678.407,E2 -678.407} C_VEL
LIN {X 0,Y 601.436,Z 396.57,A -85,B 0,C 180,E1 -681.529,E2 -681.529} C_VEL
LIN {X 0,Y 601.39,Z 396.576,A -85,B 0,C 180,E1 -684.245,E2 -684.245} C_VEL
LIN {X 0,Y 601.431,Z 396.57,A -85,B 0,C 180,E1 -686.687,E2 -686.687} C_VEL
LIN {X 0,Y 601.426,Z 396.572,A -85,B 0,C 180,E1 -689.058,E2 -689.058} C_VEL
LIN {X 0,Y 601.437,Z 396.572,A -85,B 0,C 180,E1 -691.373,E2 -691.373} C_VEL
LIN {X 0,Y 601.404,Z 396.575,A -85,B 0,C 180,E1 -693.636,E2 -693.636} C_VEL
LIN {X 0,Y 601.454,Z 396.568,A -85,B 0,C 180,E1 -695.859,E2 -695.859} C_VEL
LIN {X 0,Y 601.411,Z 396.575,A -85,B 0,C 180,E1 -698.761,E2 -698.761} C_VEL
LIN {X 0,Y 601.425,Z 396.571,A -85,B 0,C 180,E1 -701.608,E2 -701.608} C_VEL
LIN {X 0,Y 601.418,Z 396.572,A -85,B 0,C 180,E1 -704.409,E2 -704.409} C_VEL
LIN {X 0,Y 601.425,Z 396.573,A -85,B 0,C 180,E1 -707.172,E2 -707.172} C_VEL
LIN {X 0,Y 601.433,Z 396.569,A -85,B 0,C 180,E1 -709.905,E2 -709.905} C_VEL
LIN {X 0,Y 601.441,Z 396.571,A -85,B 0,C 180,E1 -712.615,E2 -712.615} C_VEL
LIN {X 0,Y 601.427,Z 396.57,A -85,B 0,C 180,E1 -715.308,E2 -715.308} C_VEL
LIN {X 0,Y 601.425,Z 396.572,A -85,B 0,C 180,E1 -717.991,E2 -717.991} C_VEL
LIN {X 0,Y 601.452,Z 396.568,A -85,B 0,C 180,E1 -720.669,E2 -720.669} C_VEL
LIN {X 0,Y 601.44,Z 396.57,A -85,B 0,C 180,E1 -723.349,E2 -723.349} C_VEL
LIN {X 0,Y 601.412,Z 396.573,A -85,B 0,C 180,E1 -726.037,E2 -726.037} C_VEL
LIN {X 0,Y 601.416,Z 396.572,A -85,B 0,C 180,E1 -728.738,E2 -728.738} C_VEL
LIN {X 0,Y 601.436,Z 396.571,A -85,B 0,C 180,E1 -731.458,E2 -731.458} C_VEL
LIN {X 0,Y 601.424,Z 396.571,A -85,B 0,C 180,E1 -734.205,E2 -734.205} C_VEL
LIN {X 0,Y 601.437,Z 396.571,A -85,B 0,C 180,E1 -736.986,E2 -736.986} C_VEL
LIN {X 0,Y 601.413,Z 396.573,A -85,B 0,C 180,E1 -739.809,E2 -739.809} C_VEL
LIN {X 0,Y 601.415,Z 396.572,A -85,B 0,C 180,E1 -742.683,E2 -742.683} C_VEL
LIN {X 0,Y 601.4,Z 396.574,A -85,B 0,C 180,E1 -744.879,E2 -744.879} C_VEL
LIN {X 0,Y 601.416,Z 396.573,A -85,B 0,C 180,E1 -747.362,E2 -747.362} C_VEL
LIN {X 0,Y 601.431,Z 396.57,A -85,B 0,C 180,E1 -750.148,E2 -750.148} C_VEL
LIN {X 0,Y 601.425,Z 396.573,A -85,B 0,C 180,E1 -752.716,E2 -752.716} C_VEL
LIN {X 0,Y 601.402,Z 396.575,A -85,B 0,C 180,E1 -755.113,E2 -755.113} C_VEL
LIN {X 0,Y 601.44,Z 396.569,A -85,B 0,C 180,E1 -757.419,E2 -757.419} C_VEL
LIN {X 0,Y 601.404,Z 396.574,A -85,B 0,C 180,E1 -759.996,E2 -759.996} C_VEL
LIN {X 0,Y 601.416,Z 396.572,A -85,B 0,C 180,E1 -762.67,E2 -762.67} C_VEL
LIN {X 0,Y 601.428,Z 396.573,A -85,B 0,C 180,E1 -765.465,E2 -765.465} C_VEL
LIN {X 0,Y 601.427,Z 396.571,A -85,B 0,C 180,E1 -768.407,E2 -768.407} C_VEL
LIN {X 0,Y 601.443,Z 396.571,A -85,B 0,C 180,E1 -770.876,E2 -770.876} C_VEL
LIN {X 0,Y 601.448,Z 396.569,A -85,B 0,C 180,E1 -773.734,E2 -773.734} C_VEL
LIN {X 0,Y 601.448,Z 396.599,A -85,B 0,C 180,E1 -774.159,E2 -774.159} C_VEL
LIN {X 0,Y 601.645,Z 403.345,A -85,B 0,C 180,E1 -775.49,E2 -775.49} C_VEL
LIN {X 0,Y 601.754,Z 419.301,A -85,B 0,C 180,E1 -778.494,E2 -778.494} C_VEL
LIN {X 0,Y 601.692,Z 432.936,A -85,B 0,C 180,E1 -781.167,E2 -781.167} C_VEL
LIN {X 0,Y 601.637,Z 448.118,A -85,B 0,C 180,E1 -784.089,E2 -784.089} C_VEL
LIN {X 0,Y 601.585,Z 463.407,A -85,B 0,C 180,E1 -786.961,E2 -786.961} C_VEL
LIN {X 0,Y 601.525,Z 479.058,A -85,B 0,C 180,E1 -789.838,E2 -789.838} C_VEL
LIN {X 0,Y 601.487,Z 492.753,A -85,B 0,C 180,E1 -792.314,E2 -792.314} C_VEL
LIN {X 0,Y 601.437,Z 508.405,A -85,B 0,C 180,E1 -795.103,E2 -795.103} C_VEL
LIN {X 0,Y 601.413,Z 525.156,A -85,B 0,C 180,E1 -798.05,E2 -798.05} C_VEL
LIN {X 0,Y 601.591,Z 537.439,A -85,B 0,C 180,E1 -798.267,E2 -798.267} C_VEL
LIN {X 0,Y 601.56,Z 550.237,A -85,B 0,C 180,E1 -798.622,E2 -798.622} C_VEL
LIN {X 0,Y 601.539,Z 561.954,A -85,B 0,C 180,E1 -799.076,E2 -799.076} C_VEL
LIN {X 0,Y 601.482,Z 573.327,A -85,B 0,C 180,E1 -799.651,E2 -799.651} C_VEL
LIN {X 0,Y 601.467,Z 583.931,A -85,B 0,C 180,E1 -800.33,E2 -800.33} C_VEL
LIN {X 0,Y 601.435,Z 593.599,A -85,B 0,C 180,E1 -801.093,E2 -801.093} C_VEL
LIN {X 0,Y 601.406,Z 602.414,A -85,B 0,C 180,E1 -801.939,E2 -801.939} C_VEL
LIN {X 0,Y 601.388,Z 609.691,A -85,B 0,C 180,E1 -802.783,E2 -802.783} C_VEL
LIN {X 0,Y 601.375,Z 616.774,A -85,B 0,C 180,E1 -803.782,E2 -803.782} C_VEL
LIN {X 0,Y 601.373,Z 621.68,A -85,B 0,C 180,E1 -804.635,E2 -804.635} C_VEL
LIN {X 0,Y 601.353,Z 626.371,A -85,B 0,C 180,E1 -805.643,E2 -805.643} C_VEL
LIN {X 0,Y 601.344,Z 629.956,A -85,B 0,C 180,E1 -806.65,E2 -806.65} C_VEL
LIN {X 0,Y 601.325,Z 631.809,A -85,B 0,C 180,E1 -807.32,E2 -807.32} C_VEL
LIN {X 0,Y 601.341,Z 633.202,A -85,B 0,C 180,E1 -807.991,E2 -807.991} C_VEL
LIN {X 0,Y 601.339,Z 634.784,A -85,B 0,C 180,E1 -809.33,E2 -809.33} C_VEL
LIN {X 0,Y 601.335,Z 635,A -85,B 0,C 180,E1 -810,E2 -810} C_VEL
LIN {X 0,Y 601.348,Z 634.184,A -85,B 0,C 180,E1 -811.339,E2 -811.339} C_VEL
LIN {X 0,Y 601.341,Z 633.202,A -85,B 0,C 180,E1 -812.009,E2 -812.009} C_VEL
LIN {X 0,Y 601.325,Z 631.809,A -85,B 0,C 180,E1 -812.68,E2 -812.68} C_VEL
LIN {X 0,Y 601.367,Z 628.896,A -85,B 0,C 180,E1 -813.685,E2 -813.685} C_VEL
LIN {X 0,Y 601.337,Z 624.949,A -85,B 0,C 180,E1 -814.693,E2 -814.693} C_VEL
LIN {X 0,Y 601.372,Z 618.876,A -85,B 0,C 180,E1 -815.869,E2 -815.869} C_VEL
LIN {X 0,Y 601.382,Z 612.235,A -85,B 0,C 180,E1 -816.88,E2 -816.88} C_VEL
LIN {X 0,Y 601.4,Z 603.988,A -85,B 0,C 180,E1 -817.892,E2 -817.892} C_VEL
LIN {X 0,Y 601.436,Z 595.535,A -85,B 0,C 180,E1 -818.738,E2 -818.738} C_VEL
LIN {X 0,Y 601.449,Z 585.09,A -85,B 0,C 180,E1 -819.585,E2 -819.585} C_VEL
LIN {X 0,Y 601.472,Z 574.755,A -85,B 0,C 180,E1 -820.265,E2 -820.265} C_VEL
LIN {X 0,Y 601.533,Z 562.644,A -85,B 0,C 180,E1 -820.894,E2 -820.894} C_VEL
LIN {X 0,Y 601.561,Z 550.223,A -85,B 0,C 180,E1 -821.378,E2 -821.378} C_VEL
LIN {X 0,Y 601.591,Z 537.433,A -85,B 0,C 180,E1 -821.733,E2 -821.733} C_VEL
LIN {X 0,Y 601.413,Z 525.156,A -85,B 0,C 180,E1 -821.95,E2 -821.95} C_VEL
LIN {X 0,Y 601.436,Z 508.404,A -85,B 0,C 180,E1 -824.897,E2 -824.897} C_VEL
LIN {X 0,Y 601.487,Z 492.752,A -85,B 0,C 180,E1 -827.686,E2 -827.686} C_VEL
LIN {X 0,Y 601.526,Z 479.057,A -85,B 0,C 180,E1 -830.162,E2 -830.162} C_VEL
LIN {X 0,Y 601.585,Z 463.406,A -85,B 0,C 180,E1 -833.039,E2 -833.039} C_VEL
LIN {X 0,Y 601.651,Z 447.215,A -85,B 0,C 180,E1 -836.082,E2 -836.082} C_VEL
LIN {X 0,Y 601.716,Z 431.789,A -85,B 0,C 180,E1 -839.056,E2 -839.056} C_VEL
LIN {X 0,Y 601.732,Z 418.2,A -85,B 0,C 180,E1 -841.708,E2 -841.708} C_VEL
LIN {X 0,Y 601.673,Z 402.304,A -85,B 0,C 180,E1 -844.711,E2 -844.711} C_VEL
LIN {X 0,Y 601.452,Z 396.57,A -85,B 0,C 180,E1 -845.863,E2 -845.863} C_VEL
LIN {X 0,Y 601.443,Z 396.569,A -85,B 0,C 180,E1 -848.472,E2 -848.472} C_VEL
LIN {X 0,Y 601.421,Z 396.571,A -85,B 0,C 180,E1 -850.874,E2 -850.874} C_VEL
LIN {X 0,Y 601.433,Z 396.571,A -85,B 0,C 180,E1 -853.586,E2 -853.586} C_VEL
LIN {X 0,Y 601.454,Z 396.568,A -85,B 0,C 180,E1 -856.425,E2 -856.425} C_VEL
LIN {X 0,Y 601.417,Z 396.572,A -85,B 0,C 180,E1 -859.427,E2 -859.427} C_VEL
LIN {X 0,Y 601.426,Z 396.572,A -85,B 0,C 180,E1 -861.732,E2 -861.732} C_VEL
LIN {X 0,Y 601.411,Z 396.573,A -85,B 0,C 180,E1 -864.247,E2 -864.247} C_VEL
LIN {X 0,Y 601.431,Z 396.57,A -85,B 0,C 180,E1 -866.687,E2 -866.687} C_VEL
LIN {X 0,Y 601.435,Z 396.57,A -85,B 0,C 180,E1 -869.059,E2 -869.059} C_VEL
LIN {X 0,Y 601.439,Z 396.571,A -85,B 0,C 180,E1 -871.373,E2 -871.373} C_VEL
LIN {X 0,Y 601.403,Z 396.576,A -85,B 0,C 180,E1 -873.636,E2 -873.636} C_VEL
LIN {X 0,Y 601.457,Z 396.568,A -85,B 0,C 180,E1 -875.86,E2 -875.86} C_VEL
LIN {X 0,Y 601.411,Z 396.574,A -85,B 0,C 180,E1 -878.761,E2 -878.761} C_VEL
LIN {X 0,Y 601.426,Z 396.571,A -85,B 0,C 180,E1 -881.608,E2 -881.608} C_VEL
LIN {X 0,Y 601.42,Z 396.572,A -85,B 0,C 180,E1 -884.409,E2 -884.409} C_VEL
LIN {X 0,Y 601.426,Z 396.572,A -85,B 0,C 180,E1 -887.172,E2 -887.172} C_VEL
LIN {X 0,Y 601.431,Z 396.57,A -85,B 0,C 180,E1 -889.905,E2 -889.905} C_VEL
LIN {X 0,Y 601.442,Z 396.571,A -85,B 0,C 180,E1 -892.615,E2 -892.615} C_VEL
LIN {X 0,Y 601.429,Z 396.57,A -85,B 0,C 180,E1 -895.308,E2 -895.308} C_VEL
LIN {X 0,Y 601.435,Z 396.572,A -85,B 0,C 180,E1 -897.991,E2 -897.991} C_VEL
LIN {X 0,Y 601.456,Z 396.567,A -85,B 0,C 180,E1 -900.67,E2 -900.67} C_VEL
LIN {X 0,Y 601.437,Z 396.571,A -85,B 0,C 180,E1 -903.35,E2 -903.35} C_VEL
LIN {X 0,Y 601.407,Z 396.573,A -85,B 0,C 180,E1 -906.037,E2 -906.037} C_VEL
LIN {X 0,Y 601.419,Z 396.573,A -85,B 0,C 180,E1 -908.738,E2 -908.738} C_VEL
LIN {X 0,Y 601.428,Z 396.571,A -85,B 0,C 180,E1 -911.458,E2 -911.458} C_VEL
LIN {X 0,Y 601.414,Z 396.572,A -85,B 0,C 180,E1 -912.374,E2 -912.374} C_VEL
LIN {X 0,Y 600.749,Z 396.657,A -85,B 0,C 180,E1 -912.933,E2 -912.933} C_VEL
LIN {X 0,Y 597.9,Z 397.013,A -85,B 0,C 180,E1 -913.841,E2 -913.841} C_VEL
LIN {X 0,Y 595.49,Z 397.312,A -85,B 0,C 180,E1 -914.571,E2 -914.571} C_VEL
LIN {X 0,Y 594.453,Z 397.441,A -85,B 0,C 180,E1 -915.135,E2 -915.135} C_VEL
LIN {X 0,Y 594.367,Z 397.45,A -85,B 0,C 180,E1 -915.326,E2 -915.326} C_VEL
LIN {X 0,Y 594.395,Z 397.448,A -85,B 0,C 180,E1 -917.193,E2 -917.193} C_VEL
LIN {X 0,Y 594.379,Z 397.45,A -85,B 0,C 180,E1 -920.054,E2 -920.054} C_VEL
LIN {X 0,Y 594.36,Z 397.451,A -85,B 0,C 180,E1 -922.968,E2 -922.968} C_VEL
LIN {X 0,Y 594.378,Z 397.449,A -85,B 0,C 180,E1 -925.193,E2 -925.193} C_VEL
LIN {X 0,Y 594.391,Z 397.449,A -85,B 0,C 180,E1 -927.527,E2 -927.527} C_VEL
LIN {X 0,Y 594.393,Z 397.446,A -85,B 0,C 180,E1 -930.329,E2 -930.329} C_VEL
LIN {X 0,Y 594.384,Z 397.451,A -85,B 0,C 180,E1 -932.95,E2 -932.95} C_VEL
LIN {X 0,Y 594.353,Z 397.452,A -85,B 0,C 180,E1 -935.409,E2 -935.409} C_VEL
LIN {X 0,Y 594.388,Z 397.448,A -85,B 0,C 180,E1 -937.941,E2 -937.941} C_VEL
LIN {X 0,Y 594.379,Z 397.448,A -85,B 0,C 180,E1 -940.822,E2 -940.822} C_VEL
LIN {X 0,Y 594.387,Z 397.447,A -85,B 0,C 180,E1 -943.841,E2 -943.841} C_VEL
LIN {X 0,Y 594.384,Z 397.451,A -85,B 0,C 180,E1 -946.702,E2 -946.702} C_VEL
LIN {X 0,Y 594.374,Z 397.449,A -85,B 0,C 180,E1 -949.433,E2 -949.433} C_VEL
LIN {X 0,Y 594.394,Z 397.447,A -85,B 0,C 180,E1 -952.391,E2 -952.391} C_VEL
LIN {X 0,Y 594.389,Z 397.448,A -85,B 0,C 180,E1 -955.42,E2 -955.42} C_VEL
LIN {X 0,Y 594.382,Z 397.451,A -85,B 0,C 180,E1 -958.357,E2 -958.357} C_VEL
LIN {X 0,Y 594.39,Z 397.447,A -85,B 0,C 180,E1 -961.042,E2 -961.042} C_VEL
LIN {X 0,Y 594.393,Z 397.447,A -85,B 0,C 180,E1 -963.977,E2 -963.977} C_VEL
LIN {X 0,Y 594.395,Z 397.446,A -85,B 0,C 180,E1 -966.296,E2 -966.296} C_VEL
LIN {X 0,Y 594.404,Z 397.446,A -85,B 0,C 180,E1 -969.224,E2 -969.224} C_VEL
LIN {X 0,Y 594.356,Z 397.454,A -85,B 0,C 180,E1 -972.095,E2 -972.095} C_VEL
LIN {X 0,Y 594.368,Z 397.452,A -85,B 0,C 180,E1 -974.219,E2 -974.219} C_VEL
LIN {X 0,Y 594.385,Z 397.45,A -85,B 0,C 180,E1 -976.321,E2 -976.321} C_VEL
LIN {X 0,Y 594.371,Z 397.452,A -85,B 0,C 180,E1 -978.425,E2 -978.425} C_VEL
LIN {X 0,Y 594.603,Z 404.01,A -85,B 0,C 180,E1 -978.665,E2 -978.665} C_VEL
LIN {X 0,Y 594.532,Z 416.015,A -85,B 0,C 180,E1 -979.184,E2 -979.184} C_VEL
LIN {X 0,Y 594.465,Z 428.237,A -85,B 0,C 180,E1 -979.871,E2 -979.871} C_VEL
LIN {X 0,Y 594.405,Z 438.981,A -85,B 0,C 180,E1 -980.644,E2 -980.644} C_VEL
LIN {X 0,Y 594.384,Z 448.648,A -85,B 0,C 180,E1 -981.5,E2 -981.5} C_VEL
LIN {X 0,Y 594.347,Z 456.578,A -85,B 0,C 180,E1 -982.355,E2 -982.355} C_VEL
LIN {X 0,Y 594.306,Z 464.399,A -85,B 0,C 180,E1 -983.39,E2 -983.39} C_VEL
LIN {X 0,Y 594.289,Z 471.446,A -85,B 0,C 180,E1 -984.571,E2 -984.571} C_VEL
LIN {X 0,Y 594.27,Z 476.188,A -85,B 0,C 180,E1 -985.591,E2 -985.591} C_VEL
LIN {X 0,Y 594.267,Z 479.82,A -85,B 0,C 180,E1 -986.61,E2 -986.61} C_VEL
LIN {X 0,Y 594.225,Z 481.693,A -85,B 0,C 180,E1 -987.288,E2 -987.288} C_VEL
LIN {X 0,Y 594.242,Z 483.13,A -85,B 0,C 180,E1 -987.967,E2 -987.967} C_VEL
LIN {X 0,Y 594.24,Z 484.753,A -85,B 0,C 180,E1 -989.322,E2 -989.322} C_VEL
LIN {X 0,Y 594.236,Z 484.996,A -85,B 0,C 180,E1 -990,E2 -990} C_VEL
LIN {X 0,Y 594.239,Z 484.815,A -85,B 0,C 180,E1 -990.678,E2 -990.678} C_VEL
LIN {X 0,Y 594.242,Z 483.276,A -85,B 0,C 180,E1 -992.033,E2 -992.033} C_VEL
LIN {X 0,Y 594.226,Z 481.915,A -85,B 0,C 180,E1 -992.712,E2 -992.712} C_VEL
LIN {X 0,Y 594.289,Z 479.043,A -85,B 0,C 180,E1 -993.729,E2 -993.729} C_VEL
LIN {X 0,Y 594.242,Z 475.144,A -85,B 0,C 180,E1 -994.749,E2 -994.749} C_VEL
LIN {X 0,Y 594.299,Z 470.112,A -85,B 0,C 180,E1 -995.769,E2 -995.769} C_VEL
LIN {X 0,Y 594.316,Z 463.783,A -85,B 0,C 180,E1 -996.791,E2 -996.791} C_VEL
LIN {X 0,Y 594.346,Z 455.874,A -85,B 0,C 180,E1 -997.816,E2 -997.816} C_VEL
LIN {X 0,Y 594.381,Z 446.021,A -85,B 0,C 180,E1 -998.842,E2 -998.842} C_VEL
LIN {X 0,Y 594.433,Z 435.702,A -85,B 0,C 180,E1 -999.699,E2 -999.699} C_VEL
LIN {X 0,Y 594.511,Z 424.084,A -85,B 0,C 180,E1 -1000.472,E2 -1000.472} C_VEL
LIN {X 0,Y 594.545,Z 412.214,A -85,B 0,C 180,E1 -1001.088,E2 -1001.088} C_VEL
LIN {X 0,Y 594.603,Z 399.25,A -85,B 0,C 180,E1 -1001.592,E2 -1001.592} C_VEL
LIN {X 0,Y 594.397,Z 397.448,A -85,B 0,C 180,E1 -1001.66,E2 -1001.66} C_VEL
LIN {X 0,Y 594.394,Z 397.446,A -85,B 0,C 180,E1 -1004.377,E2 -1004.377} C_VEL
LIN {X 0,Y 594.382,Z 397.449,A -85,B 0,C 180,E1 -1007.194,E2 -1007.194} C_VEL
LIN {X 0,Y 594.377,Z 397.452,A -85,B 0,C 180,E1 -1010.054,E2 -1010.054} C_VEL
LIN {X 0,Y 594.369,Z 397.45,A -85,B 0,C 180,E1 -1012.967,E2 -1012.967} C_VEL
LIN {X 0,Y 594.382,Z 397.449,A -85,B 0,C 180,E1 -1015.193,E2 -1015.193} C_VEL
LIN {X 0,Y 594.39,Z 397.449,A -85,B 0,C 180,E1 -1017.527,E2 -1017.527} C_VEL
LIN {X 0,Y 594.39,Z 397.447,A -85,B 0,C 180,E1 -1020.328,E2 -1020.328} C_VEL
LIN {X 0,Y 594.379,Z 397.45,A -85,B 0,C 180,E1 -1022.95,E2 -1022.95} C_VEL
LIN {X 0,Y 594.384,Z 397.448,A -85,B 0,C 180,E1 -1025.407,E2 -1025.407} C_VEL
LIN {X 0,Y 594.392,Z 397.448,A -85,B 0,C 180,E1 -1027.94,E2 -1027.94} C_VEL
LIN {X 0,Y 594.382,Z 397.448,A -85,B 0,C 180,E1 -1030.822,E2 -1030.822} C_VEL
LIN {X 0,Y 594.386,Z 397.447,A -85,B 0,C 180,E1 -1033.841,E2 -1033.841} C_VEL
LIN {X 0,Y 594.384,Z 397.449,A -85,B 0,C 180,E1 -1036.702,E2 -1036.702} C_VEL
LIN {X 0,Y 594.369,Z 397.45,A -85,B 0,C 180,E1 -1039.433,E2 -1039.433} C_VEL
LIN {X 0,Y 594.394,Z 397.446,A -85,B 0,C 180,E1 -1042.391,E2 -1042.391} C_VEL
LIN {X 0,Y 594.386,Z 397.447,A -85,B 0,C 180,E1 -1045.42,E2 -1045.42} C_VEL
LIN {X 0,Y 594.389,Z 397.449,A -85,B 0,C 180,E1 -1048.356,E2 -1048.356} C_VEL
LIN {X 0,Y 594.388,Z 397.448,A -85,B 0,C 180,E1 -1051.042,E2 -1051.042} C_VEL
LIN {X 0,Y 594.387,Z 397.447,A -85,B 0,C 180,E1 -1053.978,E2 -1053.978} C_VEL
LIN {X 0,Y 594.376,Z 397.449,A -85,B 0,C 180,E1 -1056.295,E2 -1056.295} C_VEL
LIN {X 0,Y 594.407,Z 397.445,A -85,B 0,C 180,E1 -1059.224,E2 -1059.224} C_VEL
LIN {X 0,Y 594.383,Z 397.45,A -85,B 0,C 180,E1 -1062.096,E2 -1062.096} C_VEL
LIN {X 0,Y 594.372,Z 397.451,A -85,B 0,C 180,E1 -1064.219,E2 -1064.219} C_VEL
LIN {X 0,Y 594.372,Z 397.45,A -85,B 0,C 180,E1 -1067.017,E2 -1067.017} C_VEL
LIN {X 0,Y 594.394,Z 397.446,A -85,B 0,C 180,E1 -1069.784,E2 -1069.784} C_VEL
LIN {X 0,Y 594.395,Z 397.449,A -85,B 0,C 180,E1 -1072.527,E2 -1072.527} C_VEL
LIN {X 0,Y 594.396,Z 397.446,A -85,B 0,C 180,E1 -1075.252,E2 -1075.252} C_VEL
LIN {X 0,Y 594.396,Z 397.448,A -85,B 0,C 180,E1 -1077.967,E2 -1077.967} C_VEL
LIN {X 0,Y 594.423,Z 397.443,A -85,B 0,C 180,E1 -1080.677,E2 -1080.677} C_VEL
LIN {X 0,Y 594.391,Z 397.448,A -85,B 0,C 180,E1 -1083.389,E2 -1083.389} C_VEL
LIN {X 0,Y 594.369,Z 397.451,A -85,B 0,C 180,E1 -1086.109,E2 -1086.109} C_VEL
LIN {X 0,Y 594.382,Z 397.448,A -85,B 0,C 180,E1 -1088.842,E2 -1088.842} C_VEL
LIN {X 0,Y 594.396,Z 397.449,A -85,B 0,C 180,E1 -1091.596,E2 -1091.596} C_VEL
LIN {X 0,Y 594.395,Z 397.447,A -85,B 0,C 180,E1 -1094.377,E2 -1094.377} C_VEL
LIN {X 0,Y 594.396,Z 397.447,A -85,B 0,C 180,E1 -1097.193,E2 -1097.193} C_VEL
LIN {X 0,Y 594.38,Z 397.451,A -85,B 0,C 180,E1 -1100.054,E2 -1100.054} C_VEL
LIN {X 0,Y 594.359,Z 397.451,A -85,B 0,C 180,E1 -1102.968,E2 -1102.968} C_VEL
LIN {X 0,Y 594.374,Z 397.45,A -85,B 0,C 180,E1 -1105.193,E2 -1105.193} C_VEL
LIN {X 0,Y 594.389,Z 397.45,A -85,B 0,C 180,E1 -1107.527,E2 -1107.527} C_VEL
LIN {X 0,Y 594.39,Z 397.447,A -85,B 0,C 180,E1 -1110.328,E2 -1110.328} C_VEL
LIN {X 0,Y 594.382,Z 397.449,A -85,B 0,C 180,E1 -1112.95,E2 -1112.95} C_VEL
LIN {X 0,Y 594.36,Z 397.451,A -85,B 0,C 180,E1 -1115.408,E2 -1115.408} C_VEL
LIN {X 0,Y 594.392,Z 397.448,A -85,B 0,C 180,E1 -1117.94,E2 -1117.94} C_VEL
LIN {X 0,Y 594.377,Z 397.448,A -85,B 0,C 180,E1 -1120.822,E2 -1120.822} C_VEL
LIN {X 0,Y 594.386,Z 397.448,A -85,B 0,C 180,E1 -1123.841,E2 -1123.841} C_VEL
LIN {X 0,Y 594.371,Z 397.451,A -85,B 0,C 180,E1 -1126.701,E2 -1126.701} C_VEL
LIN {X 0,Y 594.375,Z 397.449,A -85,B 0,C 180,E1 -1129.433,E2 -1129.433} C_VEL
LIN {X 0,Y 594.395,Z 397.447,A -85,B 0,C 180,E1 -1132.391,E2 -1132.391} C_VEL
LIN {X 0,Y 594.408,Z 397.491,A -85,B 0,C 180,E1 -1133.969,E2 -1133.969} C_VEL
LIN {X 0,Y 594.777,Z 402.773,A -85,B 0,C 180,E1 -1135.034,E2 -1135.034} C_VEL
LIN {X 0,Y 594.771,Z 418.9,A -85,B 0,C 180,E1 -1138.126,E2 -1138.126} C_VEL
LIN {X 0,Y 594.849,Z 430.147,A -85,B 0,C 180,E1 -1140.25,E2 -1140.25} C_VEL
LIN {X 0,Y 594.735,Z 443.842,A -85,B 0,C 180,E1 -1142.938,E2 -1142.938} C_VEL
LIN {X 0,Y 594.632,Z 457.537,A -85,B 0,C 180,E1 -1145.564,E2 -1145.564} C_VEL
LIN {X 0,Y 594.579,Z 471.232,A -85,B 0,C 180,E1 -1148.14,E2 -1148.14} C_VEL
LIN {X 0,Y 594.52,Z 486.905,A -85,B 0,C 180,E1 -1151.033,E2 -1151.033} C_VEL
LIN {X 0,Y 594.404,Z 502.535,A -85,B 0,C 180,E1 -1153.868,E2 -1153.868} C_VEL
LIN {X 0,Y 594.363,Z 518.187,A -85,B 0,C 180,E1 -1156.669,E2 -1156.669} C_VEL
LIN {X 0,Y 594.356,Z 525.156,A -85,B 0,C 180,E1 -1157.906,E2 -1157.906} C_VEL
LIN {X 0,Y 594.673,Z 530.946,A -85,B 0,C 180,E1 -1157.999,E2 -1157.999} C_VEL
LIN {X 0,Y 594.623,Z 544.217,A -85,B 0,C 180,E1 -1158.301,E2 -1158.301} C_VEL
LIN {X 0,Y 594.562,Z 557.248,A -85,B 0,C 180,E1 -1158.744,E2 -1158.744} C_VEL
LIN {X 0,Y 594.525,Z 568.633,A -85,B 0,C 180,E1 -1159.27,E2 -1159.27} C_VEL
LIN {X 0,Y 594.469,Z 580.199,A -85,B 0,C 180,E1 -1159.957,E2 -1159.957} C_VEL
LIN {X 0,Y 594.414,Z 590.596,A -85,B 0,C 180,E1 -1160.73,E2 -1160.73} C_VEL
LIN {X 0,Y 594.383,Z 599.112,A -85,B 0,C 180,E1 -1161.501,E2 -1161.501} C_VEL
LIN {X 0,Y 594.347,Z 606.961,A -85,B 0,C 180,E1 -1162.355,E2 -1162.355} C_VEL
LIN {X 0,Y 594.283,Z 614.813,A -85,B 0,C 180,E1 -1163.408,E2 -1163.408} C_VEL
LIN {X 0,Y 594.289,Z 621.68,A -85,B 0,C 180,E1 -1164.571,E2 -1164.571} C_VEL
LIN {X 0,Y 594.27,Z 626.371,A -85,B 0,C 180,E1 -1165.591,E2 -1165.591} C_VEL
LIN {X 0,Y 594.267,Z 629.956,A -85,B 0,C 180,E1 -1166.61,E2 -1166.61} C_VEL
LIN {X 0,Y 594.226,Z 631.809,A -85,B 0,C 180,E1 -1167.288,E2 -1167.288} C_VEL
LIN {X 0,Y 594.24,Z 633.202,A -85,B 0,C 180,E1 -1167.967,E2 -1167.967} C_VEL
LIN {X 0,Y 594.239,Z 634.784,A -85,B 0,C 180,E1 -1169.322,E2 -1169.322} C_VEL
LIN {X 0,Y 594.236,Z 635,A -85,B 0,C 180,E1 -1170,E2 -1170} C_VEL
LIN {X 0,Y 594.247,Z 634.185,A -85,B 0,C 180,E1 -1171.355,E2 -1171.355} C_VEL
LIN {X 0,Y 594.24,Z 633.202,A -85,B 0,C 180,E1 -1172.033,E2 -1172.033} C_VEL
LIN {X 0,Y 594.226,Z 631.809,A -85,B 0,C 180,E1 -1172.712,E2 -1172.712} C_VEL
LIN {X 0,Y 594.288,Z 628.896,A -85,B 0,C 180,E1 -1173.729,E2 -1173.729} C_VEL
LIN {X 0,Y 594.242,Z 624.949,A -85,B 0,C 180,E1 -1174.749,E2 -1174.749} C_VEL
LIN {X 0,Y 594.304,Z 618.877,A -85,B 0,C 180,E1 -1175.939,E2 -1175.939} C_VEL
LIN {X 0,Y 594.308,Z 612.235,A -85,B 0,C 180,E1 -1176.962,E2 -1176.962} C_VEL
LIN {X 0,Y 594.359,Z 603.989,A -85,B 0,C 180,E1 -1177.986,E2 -1177.986} C_VEL
LIN {X 0,Y 594.382,Z 595.536,A -85,B 0,C 180,E1 -1178.842,E2 -1178.842} C_VEL
LIN {X 0,Y 594.431,Z 585.092,A -85,B 0,C 180,E1 -1179.699,E2 -1179.699} C_VEL
LIN {X 0,Y 594.482,Z 574.756,A -85,B 0,C 180,E1 -1180.387,E2 -1180.387} C_VEL
LIN {X 0,Y 594.533,Z 563.758,A -85,B 0,C 180,E1 -1180.972,E2 -1180.972} C_VEL
LIN {X 0,Y 594.582,Z 551.718,A -85,B 0,C 180,E1 -1181.464,E2 -1181.464} C_VEL
LIN {X 0,Y 594.629,Z 538.346,A -85,B 0,C 180,E1 -1181.851,E2 -1181.851} C_VEL
LIN {X 0,Y 594.577,Z 526.593,A -85,B 0,C 180,E1 -1182.068,E2 -1182.068} C_VEL
LIN {X 0,Y 594.361,Z 525.034,A -85,B 0,C 180,E1 -1182.116,E2 -1182.116} C_VEL
LIN {X 0,Y 594.395,Z 510.36,A -85,B 0,C 180,E1 -1184.727,E2 -1184.727} C_VEL
LIN {X 0,Y 594.463,Z 494.709,A -85,B 0,C 180,E1 -1187.546,E2 -1187.546} C_VEL
LIN {X 0,Y 594.544,Z 481.014,A -85,B 0,C 180,E1 -1190.048,E2 -1190.048} C_VEL
LIN {X 0,Y 594.622,Z 465.362,A -85,B 0,C 180,E1 -1192.957,E2 -1192.957} C_VEL
LIN {X 0,Y 594.698,Z 449.711,A -85,B 0,C 180,E1 -1195.929,E2 -1195.929} C_VEL
LIN {X 0,Y 594.8,Z 436.016,A -85,B 0,C 180,E1 -1198.59,E2 -1198.59} C_VEL
LIN {X 0,Y 594.835,Z 424.997,A -85,B 0,C 180,E1 -1200.731,E2 -1200.731} C_VEL
LIN {X 0,Y 594.713,Z 410.099,A -85,B 0,C 180,E1 -1203.536,E2 -1203.536} C_VEL
LIN {X 0,Y 594.705,Z 399.604,A -85,B 0,C 180,E1 -1205.593,E2 -1205.593} C_VEL
LIN {X 0,Y 594.424,Z 397.446,A -85,B 0,C 180,E1 -1206.082,E2 -1206.082} C_VEL
LIN {X 0,Y 594.394,Z 397.447,A -85,B 0,C 180,E1 -1208.805,E2 -1208.805} C_VEL
LIN {X 0,Y 594.385,Z 397.447,A -85,B 0,C 180,E1 -1211.848,E2 -1211.848} C_VEL
LIN {X 0,Y 594.367,Z 397.45,A -85,B 0,C 180,E1 -1214.809,E2 -1214.809} C_VEL
LIN {X 0,Y 594.374,Z 397.452,A -85,B 0,C 180,E1 -1217.625,E2 -1217.625} C_VEL
LIN {X 0,Y 594.376,Z 397.449,A -85,B 0,C 180,E1 -1220.319,E2 -1220.319} C_VEL
LIN {X 0,Y 594.391,Z 397.449,A -85,B 0,C 180,E1 -1222.914,E2 -1222.914} C_VEL
LIN {X 0,Y 594.384,Z 397.448,A -85,B 0,C 180,E1 -1225.862,E2 -1225.862} C_VEL
LIN {X 0,Y 594.395,Z 397.446,A -85,B 0,C 180,E1 -1228.651,E2 -1228.651} C_VEL
LIN {X 0,Y 594.388,Z 397.447,A -85,B 0,C 180,E1 -1231.042,E2 -1231.042} C_VEL
LIN {X 0,Y 594.385,Z 397.448,A -85,B 0,C 180,E1 -1233.978,E2 -1233.978} C_VEL
LIN {X 0,Y 594.379,Z 397.448,A -85,B 0,C 180,E1 -1236.295,E2 -1236.295} C_VEL
LIN {X 0,Y 594.406,Z 397.445,A -85,B 0,C 180,E1 -1239.224,E2 -1239.224} C_VEL
LIN {X 0,Y 594.386,Z 397.45,A -85,B 0,C 180,E1 -1242.096,E2 -1242.096} C_VEL
LIN {X 0,Y 594.373,Z 397.451,A -85,B 0,C 180,E1 -1244.219,E2 -1244.219} C_VEL
LIN {X 0,Y 594.372,Z 397.449,A -85,B 0,C 180,E1 -1247.017,E2 -1247.017} C_VEL
LIN {X 0,Y 594.392,Z 397.447,A -85,B 0,C 180,E1 -1249.784,E2 -1249.784} C_VEL
LIN {X 0,Y 594.396,Z 397.448,A -85,B 0,C 180,E1 -1252.527,E2 -1252.527} C_VEL
LIN {X 0,Y 594.399,Z 397.446,A -85,B 0,C 180,E1 -1255.252,E2 -1255.252} C_VEL
LIN {X 0,Y 594.405,Z 397.448,A -85,B 0,C 180,E1 -1257.967,E2 -1257.967} C_VEL
LIN {X 0,Y 594.427,Z 397.442,A -85,B 0,C 180,E1 -1260.677,E2 -1260.677} C_VEL
LIN {X 0,Y 594.388,Z 397.449,A -85,B 0,C 180,E1 -1263.389,E2 -1263.389} C_VEL
LIN {X 0,Y 594.364,Z 397.451,A -85,B 0,C 180,E1 -1266.109,E2 -1266.109} C_VEL
LIN {X 0,Y 594.385,Z 397.448,A -85,B 0,C 180,E1 -1268.842,E2 -1268.842} C_VEL
LIN {X 0,Y 594.392,Z 397.448,A -85,B 0,C 180,E1 -1271.596,E2 -1271.596} C_VEL
LIN {X 0,Y 594.396,Z 397.446,A -85,B 0,C 180,E1 -1274.377,E2 -1274.377} C_VEL
LIN {X 0,Y 594.367,Z 397.45,A -85,B 0,C 180,E1 -1275.326,E2 -1275.326} C_VEL
LIN {X 0,Y 593.692,Z 397.536,A -85,B 0,C 180,E1 -1275.892,E2 -1275.892} C_VEL
LIN {X 0,Y 590.825,Z 397.894,A -85,B 0,C 180,E1 -1276.81,E2 -1276.81} C_VEL
LIN {X 0,Y 588.415,Z 398.195,A -85,B 0,C 180,E1 -1277.548,E2 -1277.548} C_VEL
LIN {X 0,Y 587.392,Z 398.321,A -85,B 0,C 180,E1 -1278.118,E2 -1278.118} C_VEL
LIN {X 0,Y 587.315,Z 398.329,A -85,B 0,C 180,E1 -1278.311,E2 -1278.311} C_VEL
LIN {X 0,Y 587.335,Z 398.327,A -85,B 0,C 180,E1 -1281.038,E2 -1281.038} C_VEL
LIN {X 0,Y 587.317,Z 398.33,A -85,B 0,C 180,E1 -1283.259,E2 -1283.259} C_VEL
LIN {X 0,Y 587.338,Z 398.328,A -85,B 0,C 180,E1 -1285.517,E2 -1285.517} C_VEL
LIN {X 0,Y 587.352,Z 398.324,A -85,B 0,C 180,E1 -1287.818,E2 -1287.818} C_VEL
LIN {X 0,Y 587.347,Z 398.324,A -85,B 0,C 180,E1 -1290.511,E2 -1290.511} C_VEL
LIN {X 0,Y 587.345,Z 398.326,A -85,B 0,C 180,E1 -1293.112,E2 -1293.112} C_VEL
LIN {X 0,Y 587.301,Z 398.33,A -85,B 0,C 180,E1 -1295.538,E2 -1295.538} C_VEL
LIN {X 0,Y 587.343,Z 398.325,A -85,B 0,C 180,E1 -1297.838,E2 -1297.838} C_VEL
LIN {X 0,Y 587.314,Z 398.33,A -85,B 0,C 180,E1 -1300.255,E2 -1300.255} C_VEL
LIN {X 0,Y 587.326,Z 398.327,A -85,B 0,C 180,E1 -1303.006,E2 -1303.006} C_VEL
LIN {X 0,Y 587.339,Z 398.326,A -85,B 0,C 180,E1 -1305.886,E2 -1305.886} C_VEL
LIN {X 0,Y 587.341,Z 398.327,A -85,B 0,C 180,E1 -1308.925,E2 -1308.925} C_VEL
LIN {X 0,Y 587.338,Z 398.325,A -85,B 0,C 180,E1 -1311.521,E2 -1311.521} C_VEL
LIN {X 0,Y 587.297,Z 398.333,A -85,B 0,C 180,E1 -1314.1,E2 -1314.1} C_VEL
LIN {X 0,Y 587.337,Z 398.326,A -85,B 0,C 180,E1 -1316.603,E2 -1316.603} C_VEL
LIN {X 0,Y 587.341,Z 398.327,A -85,B 0,C 180,E1 -1319.49,E2 -1319.49} C_VEL
LIN {X 0,Y 587.356,Z 398.323,A -85,B 0,C 180,E1 -1322.307,E2 -1322.307} C_VEL
LIN {X 0,Y 587.341,Z 398.326,A -85,B 0,C 180,E1 -1324.483,E2 -1324.483} C_VEL
LIN {X 0,Y 587.323,Z 398.328,A -85,B 0,C 180,E1 -1327.131,E2 -1327.131} C_VEL
LIN {X 0,Y 587.329,Z 398.327,A -85,B 0,C 180,E1 -1329.695,E2 -1329.695} C_VEL
LIN {X 0,Y 587.35,Z 398.324,A -85,B 0,C 180,E1 -1332.594,E2 -1332.594} C_VEL
LIN {X 0,Y 587.37,Z 398.322,A -85,B 0,C 180,E1 -1335.739,E2 -1335.739} C_VEL
LIN {X 0,Y 587.36,Z 398.324,A -85,B 0,C 180,E1 -1338.309,E2 -1338.309} C_VEL
LIN {X 0,Y 587.645,Z 403.271,A -85,B 0,C 180,E1 -1338.5,E2 -1338.5} C_VEL
LIN {X 0,Y 587.553,Z 416.03,A -85,B 0,C 180,E1 -1339.054,E2 -1339.054} C_VEL
LIN {X 0,Y 587.451,Z 428.245,A -85,B 0,C 180,E1 -1339.749,E2 -1339.749} C_VEL
LIN {X 0,Y 587.382,Z 438.989,A -85,B 0,C 180,E1 -1340.531,E2 -1340.531} C_VEL
LIN {X 0,Y 587.323,Z 448.656,A -85,B 0,C 180,E1 -1341.397,E2 -1341.397} C_VEL
LIN {X 0,Y 587.274,Z 456.584,A -85,B 0,C 180,E1 -1342.263,E2 -1342.263} C_VEL
LIN {X 0,Y 587.247,Z 464.833,A -85,B 0,C 180,E1 -1343.376,E2 -1343.376} C_VEL
LIN {X 0,Y 587.211,Z 471.452,A -85,B 0,C 180,E1 -1344.506,E2 -1344.506} C_VEL
LIN {X 0,Y 587.188,Z 476.193,A -85,B 0,C 180,E1 -1345.538,E2 -1345.538} C_VEL
LIN {X 0,Y 587.193,Z 479.824,A -85,B 0,C 180,E1 -1346.569,E2 -1346.569} C_VEL
LIN {X 0,Y 587.131,Z 481.693,A -85,B 0,C 180,E1 -1347.256,E2 -1347.256} C_VEL
LIN {X 0,Y 587.14,Z 483.132,A -85,B 0,C 180,E1 -1347.942,E2 -1347.942} C_VEL
LIN {X 0,Y 587.14,Z 484.754,A -85,B 0,C 180,E1 -1349.314,E2 -1349.314} C_VEL
LIN {X 0,Y 587.137,Z 484.996,A -85,B 0,C 180,E1 -1350,E2 -1350} C_VEL
LIN {X 0,Y 587.14,Z 484.814,A -85,B 0,C 180,E1 -1350.686,E2 -1350.686} C_VEL
LIN {X 0,Y 587.141,Z 483.276,A -85,B 0,C 180,E1 -1352.058,E2 -1352.058} C_VEL
LIN {X 0,Y 587.133,Z 481.913,A -85,B 0,C 180,E1 -1352.744,E2 -1352.744} C_VEL
LIN {X 0,Y 587.213,Z 479.042,A -85,B 0,C 180,E1 -1353.774,E2 -1353.774} C_VEL
LIN {X 0,Y 587.147,Z 475.144,A -85,B 0,C 180,E1 -1354.806,E2 -1354.806} C_VEL
LIN {X 0,Y 587.229,Z 470.108,A -85,B 0,C 180,E1 -1355.839,E2 -1355.839} C_VEL
LIN {X 0,Y 587.23,Z 463.777,A -85,B 0,C 180,E1 -1356.874,E2 -1356.874} C_VEL
LIN {X 0,Y 587.288,Z 455.872,A -85,B 0,C 180,E1 -1357.91,E2 -1357.91} C_VEL
LIN {X 0,Y 587.343,Z 446.014,A -85,B 0,C 180,E1 -1358.949,E2 -1358.949} C_VEL
LIN {X 0,Y 587.421,Z 435.696,A -85,B 0,C 180,E1 -1359.816,E2 -1359.816} C_VEL
LIN {X 0,Y 587.523,Z 424.076,A -85,B 0,C 180,E1 -1360.598,E2 -1360.598} C_VEL
LIN {X 0,Y 587.57,Z 411.768,A -85,B 0,C 180,E1 -1361.241,E2 -1361.241} C_VEL
LIN {X 0,Y 587.522,Z 399.241,A -85,B 0,C 180,E1 -1361.733,E2 -1361.733} C_VEL
LIN {X 0,Y 587.363,Z 398.324,A -85,B 0,C 180,E1 -1361.78,E2 -1361.78} C_VEL
LIN {X 0,Y 587.343,Z 398.324,A -85,B 0,C 180,E1 -1364.553,E2 -1364.553} C_VEL
LIN {X 0,Y 587.347,Z 398.324,A -85,B 0,C 180,E1 -1367.406,E2 -1367.406} C_VEL
LIN {X 0,Y 587.332,Z 398.327,A -85,B 0,C 180,E1 -1370.305,E2 -1370.305} C_VEL
LIN {X 0,Y 587.328,Z 398.329,A -85,B 0,C 180,E1 -1373.259,E2 -1373.259} C_VEL
LIN {X 0,Y 587.342,Z 398.326,A -85,B 0,C 180,E1 -1375.516,E2 -1375.516} C_VEL
LIN {X 0,Y 587.354,Z 398.324,A -85,B 0,C 180,E1 -1377.817,E2 -1377.817} C_VEL
LIN {X 0,Y 587.34,Z 398.326,A -85,B 0,C 180,E1 -1380.51,E2 -1380.51} C_VEL
LIN {X 0,Y 587.336,Z 398.326,A -85,B 0,C 180,E1 -1383.397,E2 -1383.397} C_VEL
LIN {X 0,Y 587.354,Z 398.326,A -85,B 0,C 180,E1 -1385.896,E2 -1385.896} C_VEL
LIN {X 0,Y 587.338,Z 398.325,A -85,B 0,C 180,E1 -1388.479,E2 -1388.479} C_VEL
LIN {X 0,Y 587.341,Z 398.327,A -85,B 0,C 180,E1 -1391.157,E2 -1391.157} C_VEL
LIN {X 0,Y 587.338,Z 398.325,A -85,B 0,C 180,E1 -1394.114,E2 -1394.114} C_VEL
LIN {X 0,Y 587.326,Z 398.327,A -85,B 0,C 180,E1 -1396.994,E2 -1396.994} C_VEL
LIN {X 0,Y 587.314,Z 398.331,A -85,B 0,C 180,E1 -1399.745,E2 -1399.745} C_VEL
LIN {X 0,Y 587.349,Z 398.324,A -85,B 0,C 180,E1 -1402.392,E2 -1402.392} C_VEL
LIN {X 0,Y 587.366,Z 398.322,A -85,B 0,C 180,E1 -1405.78,E2 -1405.78} C_VEL
LIN {X 0,Y 587.352,Z 398.326,A -85,B 0,C 180,E1 -1408.232,E2 -1408.232} C_VEL
LIN {X 0,Y 587.354,Z 398.323,A -85,B 0,C 180,E1 -1410.866,E2 -1410.866} C_VEL
LIN {X 0,Y 587.362,Z 398.323,A -85,B 0,C 180,E1 -1413.819,E2 -1413.819} C_VEL
LIN {X 0,Y 587.33,Z 398.326,A -85,B 0,C 180,E1 -1415.993,E2 -1415.993} C_VEL
LIN {X 0,Y 587.327,Z 398.327,A -85,B 0,C 180,E1 -1418.226,E2 -1418.226} C_VEL
LIN {X 0,Y 587.354,Z 398.324,A -85,B 0,C 180,E1 -1421.151,E2 -1421.151} C_VEL
LIN {X 0,Y 587.357,Z 398.323,A -85,B 0,C 180,E1 -1423.311,E2 -1423.311} C_VEL
LIN {X 0,Y 587.364,Z 398.324,A -85,B 0,C 180,E1 -1426.154,E2 -1426.154} C_VEL
LIN {X 0,Y 587.346,Z 398.325,A -85,B 0,C 180,E1 -1428.962,E2 -1428.962} C_VEL
LIN {X 0,Y 587.344,Z 398.325,A -85,B 0,C 180,E1 -1431.744,E2 -1431.744} C_VEL
LIN {X 0,Y 587.361,Z 398.324,A -85,B 0,C 180,E1 -1434.507,E2 -1434.507} C_VEL
LIN {X 0,Y 587.381,Z 398.32,A -85,B 0,C 180,E1 -1437.257,E2 -1437.257} C_VEL
LIN {X 0,Y 587.387,Z 398.322,A -85,B 0,C 180,E1 -1440,E2 -1440} C_VEL
LIN {X 0,Y 587.38,Z 398.32,A -85,B 0,C 180,E1 -1442.743,E2 -1442.743} C_VEL
LIN {X 0,Y 587.364,Z 398.323,A -85,B 0,C 180,E1 -1445.493,E2 -1445.493} C_VEL
LIN {X 0,Y 587.344,Z 398.326,A -85,B 0,C 180,E1 -1448.256,E2 -1448.256} C_VEL
LIN {X 0,Y 587.352,Z 398.323,A -85,B 0,C 180,E1 -1451.134,E2 -1451.134} C_VEL
LIN {X 0,Y 587.369,Z 398.322,A -85,B 0,C 180,E1 -1454.261,E2 -1454.261} C_VEL
LIN {X 0,Y 587.363,Z 398.322,A -85,B 0,C 180,E1 -1457.406,E2 -1457.406} C_VEL
LIN {X 0,Y 587.334,Z 398.327,A -85,B 0,C 180,E1 -1460.305,E2 -1460.305} C_VEL
LIN {X 0,Y 587.316,Z 398.33,A -85,B 0,C 180,E1 -1463.259,E2 -1463.259} C_VEL
LIN {X 0,Y 587.334,Z 398.328,A -85,B 0,C 180,E1 -1465.517,E2 -1465.517} C_VEL
LIN {X 0,Y 587.351,Z 398.324,A -85,B 0,C 180,E1 -1467.818,E2 -1467.818} C_VEL
LIN {X 0,Y 587.345,Z 398.326,A -85,B 0,C 180,E1 -1470.511,E2 -1470.511} C_VEL
LIN {X 0,Y 587.343,Z 398.325,A -85,B 0,C 180,E1 -1473.112,E2 -1473.112} C_VEL
LIN {X 0,Y 587.351,Z 398.326,A -85,B 0,C 180,E1 -1475.896,E2 -1475.896} C_VEL
LIN {X 0,Y 587.334,Z 398.326,A -85,B 0,C 180,E1 -1478.479,E2 -1478.479} C_VEL
LIN {X 0,Y 587.338,Z 398.327,A -85,B 0,C 180,E1 -1481.157,E2 -1481.157} C_VEL
LIN {X 0,Y 587.338,Z 398.326,A -85,B 0,C 180,E1 -1484.114,E2 -1484.114} C_VEL
LIN {X 0,Y 587.319,Z 398.328,A -85,B 0,C 180,E1 -1486.994,E2 -1486.994} C_VEL
LIN {X 0,Y 587.323,Z 398.33,A -85,B 0,C 180,E1 -1489.746,E2 -1489.746} C_VEL
LIN {X 0,Y 587.35,Z 398.325,A -85,B 0,C 180,E1 -1492.393,E2 -1492.393} C_VEL
LIN {X 0,Y 587.396,Z 398.423,A -85,B 0,C 180,E1 -1493.789,E2 -1493.789} C_VEL
LIN {X 0,Y 587.869,Z 402.757,A -85,B 0,C 180,E1 -1494.692,E2 -1494.692} C_VEL
LIN {X 0,Y 587.807,Z 418.769,A -85,B 0,C 180,E1 -1497.811,E2 -1497.811} C_VEL
LIN {X 0,Y 587.918,Z 433.907,A -85,B 0,C 180,E1 -1500.652,E2 -1500.652} C_VEL
LIN {X 0,Y 587.798,Z 447.757,A -85,B 0,C 180,E1 -1503.361,E2 -1503.361} C_VEL
LIN {X 0,Y 587.698,Z 461.45,A -85,B 0,C 180,E1 -1506.009,E2 -1506.009} C_VEL
LIN {X 0,Y 587.568,Z 475.147,A -85,B 0,C 180,E1 -1508.604,E2 -1508.604} C_VEL
LIN {X 0,Y 587.494,Z 488.84,A -85,B 0,C 180,E1 -1511.156,E2 -1511.156} C_VEL
LIN {X 0,Y 587.401,Z 502.535,A -85,B 0,C 180,E1 -1513.67,E2 -1513.67} C_VEL
LIN {X 0,Y 587.341,Z 518.187,A -85,B 0,C 180,E1 -1516.507,E2 -1516.507} C_VEL
LIN {X 0,Y 587.315,Z 525.156,A -85,B 0,C 180,E1 -1517.759,E2 -1517.759} C_VEL
LIN {X 0,Y 587.744,Z 530.946,A -85,B 0,C 180,E1 -1517.855,E2 -1517.855} C_VEL
LIN {X 0,Y 587.671,Z 544.218,A -85,B 0,C 180,E1 -1518.16,E2 -1518.16} C_VEL
LIN {X 0,Y 587.623,Z 556.663,A -85,B 0,C 180,E1 -1518.587,E2 -1518.587} C_VEL
LIN {X 0,Y 587.527,Z 568.632,A -85,B 0,C 180,E1 -1519.14,E2 -1519.14} C_VEL
LIN {X 0,Y 587.448,Z 580.201,A -85,B 0,C 180,E1 -1519.836,E2 -1519.836} C_VEL
LIN {X 0,Y 587.367,Z 590.597,A -85,B 0,C 180,E1 -1520.617,E2 -1520.617} C_VEL
LIN {X 0,Y 587.321,Z 599.112,A -85,B 0,C 180,E1 -1521.398,E2 -1521.398} C_VEL
LIN {X 0,Y 587.274,Z 606.961,A -85,B 0,C 180,E1 -1522.263,E2 -1522.263} C_VEL
LIN {X 0,Y 587.23,Z 613.47,A -85,B 0,C 180,E1 -1523.126,E2 -1523.126} C_VEL
LIN {X 0,Y 587.236,Z 619.866,A -85,B 0,C 180,E1 -1524.161,E2 -1524.161} C_VEL
LIN {X 0,Y 587.147,Z 624.95,A -85,B 0,C 180,E1 -1525.194,E2 -1525.194} C_VEL
LIN {X 0,Y 587.212,Z 628.896,A -85,B 0,C 180,E1 -1526.226,E2 -1526.226} C_VEL
LIN {X 0,Y 587.132,Z 631.809,A -85,B 0,C 180,E1 -1527.256,E2 -1527.256} C_VEL
LIN {X 0,Y 587.139,Z 633.201,A -85,B 0,C 180,E1 -1527.942,E2 -1527.942} C_VEL
LIN {X 0,Y 587.14,Z 634.784,A -85,B 0,C 180,E1 -1529.314,E2 -1529.314} C_VEL
LIN {X 0,Y 587.137,Z 635,A -85,B 0,C 180,E1 -1530,E2 -1530} C_VEL
LIN {X 0,Y 587.147,Z 634.185,A -85,B 0,C 180,E1 -1531.372,E2 -1531.372} C_VEL
LIN {X 0,Y 587.139,Z 633.201,A -85,B 0,C 180,E1 -1532.058,E2 -1532.058} C_VEL
LIN {X 0,Y 587.132,Z 631.809,A -85,B 0,C 180,E1 -1532.744,E2 -1532.744} C_VEL
LIN {X 0,Y 587.212,Z 628.896,A -85,B 0,C 180,E1 -1533.774,E2 -1533.774} C_VEL
LIN {X 0,Y 587.147,Z 624.949,A -85,B 0,C 180,E1 -1534.806,E2 -1534.806} C_VEL
LIN {X 0,Y 587.217,Z 618.877,A -85,B 0,C 180,E1 -1536.011,E2 -1536.011} C_VEL
LIN {X 0,Y 587.245,Z 612.236,A -85,B 0,C 180,E1 -1537.046,E2 -1537.046} C_VEL
LIN {X 0,Y 587.299,Z 603.989,A -85,B 0,C 180,E1 -1538.083,E2 -1538.083} C_VEL
LIN {X 0,Y 587.343,Z 595.536,A -85,B 0,C 180,E1 -1538.949,E2 -1538.949} C_VEL
LIN {X 0,Y 587.417,Z 585.093,A -85,B 0,C 180,E1 -1539.816,E2 -1539.816} C_VEL
LIN {X 0,Y 587.501,Z 574.757,A -85,B 0,C 180,E1 -1540.511,E2 -1540.511} C_VEL
LIN {X 0,Y 587.56,Z 562.829,A -85,B 0,C 180,E1 -1541.148,E2 -1541.148} C_VEL
LIN {X 0,Y 587.624,Z 550.603,A -85,B 0,C 180,E1 -1541.639,E2 -1541.639} C_VEL
LIN {X 0,Y 587.712,Z 537.431,A -85,B 0,C 180,E1 -1542.014,E2 -1542.014} C_VEL
LIN {X 0,Y 587.52,Z 526.593,A -85,B 0,C 180,E1 -1542.215,E2 -1542.215} C_VEL
LIN {X 0,Y 587.32,Z 525.034,A -85,B 0,C 180,E1 -1542.263,E2 -1542.263} C_VEL
LIN {X 0,Y 587.359,Z 510.36,A -85,B 0,C 180,E1 -1544.907,E2 -1544.907} C_VEL
LIN {X 0,Y 587.459,Z 494.709,A -85,B 0,C 180,E1 -1547.762,E2 -1547.762} C_VEL
LIN {X 0,Y 587.554,Z 479.057,A -85,B 0,C 180,E1 -1550.663,E2 -1550.663} C_VEL
LIN {X 0,Y 587.649,Z 465.362,A -85,B 0,C 180,E1 -1553.245,E2 -1553.245} C_VEL
LIN {X 0,Y 587.764,Z 451.667,A -85,B 0,C 180,E1 -1555.877,E2 -1555.877} C_VEL
LIN {X 0,Y 587.887,Z 437.972,A -85,B 0,C 180,E1 -1558.567,E2 -1558.567} C_VEL
LIN {X 0,Y 587.846,Z 424.323,A -85,B 0,C 180,E1 -1561.137,E2 -1561.137} C_VEL
LIN {X 0,Y 587.778,Z 409.472,A -85,B 0,C 180,E1 -1563.986,E2 -1563.986} C_VEL
LIN {X 0,Y 587.805,Z 401.284,A -85,B 0,C 180,E1 -1565.606,E2 -1565.606} C_VEL
LIN {X 0,Y 587.365,Z 398.324,A -85,B 0,C 180,E1 -1566.266,E2 -1566.266} C_VEL
LIN {X 0,Y 587.341,Z 398.326,A -85,B 0,C 180,E1 -1568.942,E2 -1568.942} C_VEL
LIN {X 0,Y 587.357,Z 398.323,A -85,B 0,C 180,E1 -1572.072,E2 -1572.072} C_VEL
LIN {X 0,Y 587.32,Z 398.328,A -85,B 0,C 180,E1 -1575.089,E2 -1575.089} C_VEL
LIN {X 0,Y 587.357,Z 398.324,A -85,B 0,C 180,E1 -1577.928,E2 -1577.928} C_VEL
LIN {X 0,Y 587.329,Z 398.327,A -85,B 0,C 180,E1 -1581.059,E2 -1581.059} C_VEL
LIN {X 0,Y 587.359,Z 398.323,A -85,B 0,C 180,E1 -1583.292,E2 -1583.292} C_VEL
LIN {X 0,Y 587.365,Z 398.322,A -85,B 0,C 180,E1 -1585.78,E2 -1585.78} C_VEL
LIN {X 0,Y 587.357,Z 398.326,A -85,B 0,C 180,E1 -1588.232,E2 -1588.232} C_VEL
LIN {X 0,Y 587.354,Z 398.323,A -85,B 0,C 180,E1 -1590.867,E2 -1590.867} C_VEL
LIN {X 0,Y 587.361,Z 398.323,A -85,B 0,C 180,E1 -1593.819,E2 -1593.819} C_VEL
LIN {X 0,Y 587.332,Z 398.327,A -85,B 0,C 180,E1 -1595.993,E2 -1595.993} C_VEL
LIN {X 0,Y 587.329,Z 398.327,A -85,B 0,C 180,E1 -1598.226,E2 -1598.226} C_VEL
LIN {X 0,Y 587.354,Z 398.325,A -85,B 0,C 180,E1 -1601.151,E2 -1601.151} C_VEL
LIN {X 0,Y 587.356,Z 398.324,A -85,B 0,C 180,E1 -1603.311,E2 -1603.311} C_VEL
LIN {X 0,Y 587.364,Z 398.324,A -85,B 0,C 180,E1 -1606.154,E2 -1606.154} C_VEL
LIN {X 0,Y 587.345,Z 398.324,A -85,B 0,C 180,E1 -1608.962,E2 -1608.962} C_VEL
LIN {X 0,Y 587.345,Z 398.326,A -85,B 0,C 180,E1 -1611.744,E2 -1611.744} C_VEL
LIN {X 0,Y 587.364,Z 398.323,A -85,B 0,C 180,E1 -1614.507,E2 -1614.507} C_VEL
LIN {X 0,Y 587.38,Z 398.32,A -85,B 0,C 180,E1 -1617.257,E2 -1617.257} C_VEL
LIN {X 0,Y 587.386,Z 398.322,A -85,B 0,C 180,E1 -1620,E2 -1620} C_VEL
LIN {X 0,Y 587.381,Z 398.32,A -85,B 0,C 180,E1 -1622.743,E2 -1622.743} C_VEL
LIN {X 0,Y 587.359,Z 398.325,A -85,B 0,C 180,E1 -1625.493,E2 -1625.493} C_VEL
LIN {X 0,Y 587.346,Z 398.325,A -85,B 0,C 180,E1 -1628.256,E2 -1628.256} C_VEL
LIN {X 0,Y 587.353,Z 398.324,A -85,B 0,C 180,E1 -1631.134,E2 -1631.134} C_VEL
LIN {X 0,Y 587.371,Z 398.321,A -85,B 0,C 180,E1 -1634.261,E2 -1634.261} C_VEL
LIN {X 0,Y 587.355,Z 398.324,A -85,B 0,C 180,E1 -1637.406,E2 -1637.406} C_VEL
LIN {X 0,Y 587.315,Z 398.329,A -85,B 0,C 180,E1 -1638.311,E2 -1638.311} C_VEL
LIN {X 0,Y 586.672,Z 398.409,A -85,B 0,C 180,E1 -1638.883,E2 -1638.883} C_VEL
LIN {X 0,Y 583.847,Z 398.764,A -85,B 0,C 180,E1 -1639.812,E2 -1639.812} C_VEL
LIN {X 0,Y 581.436,Z 399.066,A -85,B 0,C 180,E1 -1640.559,E2 -1640.559} C_VEL
LIN {X 0,Y 580.383,Z 399.196,A -85,B 0,C 180,E1 -1641.135,E2 -1641.135} C_VEL
LIN {X 0,Y 580.288,Z 399.206,A -85,B 0,C 180,E1 -1641.331,E2 -1641.331} C_VEL
LIN {X 0,Y 580.301,Z 399.204,A -85,B 0,C 180,E1 -1644.316,E2 -1644.316} C_VEL
LIN {X 0,Y 580.282,Z 399.207,A -85,B 0,C 180,E1 -1646.623,E2 -1646.623} C_VEL
LIN {X 0,Y 580.308,Z 399.201,A -85,B 0,C 180,E1 -1649.31,E2 -1649.31} C_VEL
LIN {X 0,Y 580.309,Z 399.201,A -85,B 0,C 180,E1 -1652.2,E2 -1652.2} C_VEL
LIN {X 0,Y 580.294,Z 399.203,A -85,B 0,C 180,E1 -1654.696,E2 -1654.696} C_VEL
LIN {X 0,Y 580.303,Z 399.204,A -85,B 0,C 180,E1 -1657.268,E2 -1657.268} C_VEL
LIN {X 0,Y 580.294,Z 399.205,A -85,B 0,C 180,E1 -1660.27,E2 -1660.27} C_VEL
LIN {X 0,Y 580.286,Z 399.205,A -85,B 0,C 180,E1 -1662.706,E2 -1662.706} C_VEL
LIN {X 0,Y 580.279,Z 399.207,A -85,B 0,C 180,E1 -1665.609,E2 -1665.609} C_VEL
LIN {X 0,Y 580.319,Z 399.199,A -85,B 0,C 180,E1 -1668.234,E2 -1668.234} C_VEL
LIN {X 0,Y 580.295,Z 399.205,A -85,B 0,C 180,E1 -1670.966,E2 -1670.966} C_VEL
LIN {X 0,Y 580.273,Z 399.205,A -85,B 0,C 180,E1 -1673.596,E2 -1673.596} C_VEL
LIN {X 0,Y 580.32,Z 399.201,A -85,B 0,C 180,E1 -1676.145,E2 -1676.145} C_VEL
LIN {X 0,Y 580.28,Z 399.205,A -85,B 0,C 180,E1 -1678.615,E2 -1678.615} C_VEL
LIN {X 0,Y 580.299,Z 399.202,A -85,B 0,C 180,E1 -1681.024,E2 -1681.024} C_VEL
LIN {X 0,Y 580.297,Z 399.205,A -85,B 0,C 180,E1 -1683.666,E2 -1683.666} C_VEL
LIN {X 0,Y 580.306,Z 399.203,A -85,B 0,C 180,E1 -1685.684,E2 -1685.684} C_VEL
LIN {X 0,Y 580.277,Z 399.207,A -85,B 0,C 180,E1 -1687.947,E2 -1687.947} C_VEL
LIN {X 0,Y 580.3,Z 399.204,A -85,B 0,C 180,E1 -1690.913,E2 -1690.913} C_VEL
LIN {X 0,Y 580.28,Z 399.204,A -85,B 0,C 180,E1 -1693.825,E2 -1693.825} C_VEL
LIN {X 0,Y 580.331,Z 399.199,A -85,B 0,C 180,E1 -1695.983,E2 -1695.983} C_VEL
LIN {X 0,Y 580.291,Z 399.204,A -85,B 0,C 180,E1 -1698.207,E2 -1698.207} C_VEL
LIN {X 0,Y 580.69,Z 402.962,A -85,B 0,C 180,E1 -1698.348,E2 -1698.348} C_VEL
LIN {X 0,Y 580.609,Z 414.296,A -85,B 0,C 180,E1 -1698.833,E2 -1698.833} C_VEL
LIN {X 0,Y 580.506,Z 425.45,A -85,B 0,C 180,E1 -1699.449,E2 -1699.449} C_VEL
LIN {X 0,Y 580.374,Z 436.823,A -85,B 0,C 180,E1 -1700.239,E2 -1700.239} C_VEL
LIN {X 0,Y 580.305,Z 446.882,A -85,B 0,C 180,E1 -1701.117,E2 -1701.117} C_VEL
LIN {X 0,Y 580.222,Z 456.59,A -85,B 0,C 180,E1 -1702.168,E2 -1702.168} C_VEL
LIN {X 0,Y 580.168,Z 464.281,A -85,B 0,C 180,E1 -1703.209,E2 -1703.209} C_VEL
LIN {X 0,Y 580.165,Z 469.612,A -85,B 0,C 180,E1 -1704.09,E2 -1704.09} C_VEL
LIN {X 0,Y 580.054,Z 474.75,A -85,B 0,C 180,E1 -1705.135,E2 -1705.135} C_VEL
LIN {X 0,Y 580.11,Z 478.74,A -85,B 0,C 180,E1 -1706.179,E2 -1706.179} C_VEL
LIN {X 0,Y 580.043,Z 481.693,A -85,B 0,C 180,E1 -1707.222,E2 -1707.222} C_VEL
LIN {X 0,Y 580.04,Z 483.134,A -85,B 0,C 180,E1 -1707.917,E2 -1707.917} C_VEL
LIN {X 0,Y 580.041,Z 484.755,A -85,B 0,C 180,E1 -1709.306,E2 -1709.306} C_VEL
LIN {X 0,Y 580.038,Z 484.996,A -85,B 0,C 180,E1 -1710,E2 -1710} C_VEL
LIN {X 0,Y 580.04,Z 484.814,A -85,B 0,C 180,E1 -1710.694,E2 -1710.694} C_VEL
LIN {X 0,Y 580.04,Z 483.275,A -85,B 0,C 180,E1 -1712.083,E2 -1712.083} C_VEL
LIN {X 0,Y 580.044,Z 481.911,A -85,B 0,C 180,E1 -1712.778,E2 -1712.778} C_VEL
LIN {X 0,Y 580.11,Z 479.041,A -85,B 0,C 180,E1 -1713.821,E2 -1713.821} C_VEL
LIN {X 0,Y 580.054,Z 475.143,A -85,B 0,C 180,E1 -1714.865,E2 -1714.865} C_VEL
LIN {X 0,Y 580.162,Z 470.102,A -85,B 0,C 180,E1 -1715.91,E2 -1715.91} C_VEL
LIN {X 0,Y 580.158,Z 463.771,A -85,B 0,C 180,E1 -1716.958,E2 -1716.958} C_VEL
LIN {X 0,Y 580.241,Z 455.869,A -85,B 0,C 180,E1 -1718.007,E2 -1718.007} C_VEL
LIN {X 0,Y 580.305,Z 447.799,A -85,B 0,C 180,E1 -1718.883,E2 -1718.883} C_VEL
LIN {X 0,Y 580.37,Z 437.952,A -85,B 0,C 180,E1 -1719.761,E2 -1719.761} C_VEL
LIN {X 0,Y 580.51,Z 426.888,A -85,B 0,C 180,E1 -1720.551,E2 -1720.551} C_VEL
LIN {X 0,Y 580.575,Z 414.393,A -85,B 0,C 180,E1 -1721.253,E2 -1721.253} C_VEL
LIN {X 0,Y 580.685,Z 402.021,A -85,B 0,C 180,E1 -1721.776,E2 -1721.776} C_VEL
LIN {X 0,Y 580.313,Z 399.201,A -85,B 0,C 180,E1 -1721.903,E2 -1721.903} C_VEL
LIN {X 0,Y 580.29,Z 399.204,A -85,B 0,C 180,E1 -1724.734,E2 -1724.734} C_VEL
LIN {X 0,Y 580.293,Z 399.203,A -85,B 0,C 180,E1 -1727.625,E2 -1727.625} C_VEL
LIN {X 0,Y 580.292,Z 399.204,A -85,B 0,C 180,E1 -1729.823,E2 -1729.823} C_VEL
LIN {X 0,Y 580.278,Z 399.207,A -85,B 0,C 180,E1 -1732.052,E2 -1732.052} C_VEL
LIN {X 0,Y 580.313,Z 399.201,A -85,B 0,C 180,E1 -1735.08,E2 -1735.08} C_VEL
LIN {X 0,Y 580.325,Z 399.199,A -85,B 0,C 180,E1 -1737.863,E2 -1737.863} C_VEL
LIN {X 0,Y 580.288,Z 399.206,A -85,B 0,C 180,E1 -1740.695,E2 -1740.695} C_VEL
LIN {X 0,Y 580.305,Z 399.202,A -85,B 0,C 180,E1 -1743.316,E2 -1743.316} C_VEL
LIN {X 0,Y 580.325,Z 399.2,A -85,B 0,C 180,E1 -1745.767,E2 -1745.767} C_VEL
LIN {X 0,Y 580.294,Z 399.205,A -85,B 0,C 180,E1 -1748.146,E2 -1748.146} C_VEL
LIN {X 0,Y 580.304,Z 399.202,A -85,B 0,C 180,E1 -1750.843,E2 -1750.843} C_VEL
LIN {X 0,Y 580.292,Z 399.203,A -85,B 0,C 180,E1 -1753.657,E2 -1753.657} C_VEL
LIN {X 0,Y 580.289,Z 399.206,A -85,B 0,C 180,E1 -1756.608,E2 -1756.608} C_VEL
LIN {X 0,Y 580.3,Z 399.202,A -85,B 0,C 180,E1 -1759.156,E2 -1759.156} C_VEL
LIN {X 0,Y 580.294,Z 399.205,A -85,B 0,C 180,E1 -1761.927,E2 -1761.927} C_VEL
LIN {X 0,Y 580.256,Z 399.208,A -85,B 0,C 180,E1 -1764.453,E2 -1764.453} C_VEL
LIN {X 0,Y 580.296,Z 399.204,A -85,B 0,C 180,E1 -1766.975,E2 -1766.975} C_VEL
LIN {X 0,Y 580.303,Z 399.202,A -85,B 0,C 180,E1 -1769.425,E2 -1769.425} C_VEL
LIN {X 0,Y 580.302,Z 399.202,A -85,B 0,C 180,E1 -1772.141,E2 -1772.141} C_VEL
LIN {X 0,Y 580.325,Z 399.199,A -85,B 0,C 180,E1 -1775.27,E2 -1775.27} C_VEL
LIN {X 0,Y 580.277,Z 399.206,A -85,B 0,C 180,E1 -1777.947,E2 -1777.947} C_VEL
LIN {X 0,Y 580.323,Z 399.202,A -85,B 0,C 180,E1 -1780.914,E2 -1780.914} C_VEL
LIN {X 0,Y 580.285,Z 399.204,A -85,B 0,C 180,E1 -1783.826,E2 -1783.826} C_VEL
LIN {X 0,Y 580.33,Z 399.199,A -85,B 0,C 180,E1 -1785.983,E2 -1785.983} C_VEL
LIN {X 0,Y 580.309,Z 399.201,A -85,B 0,C 180,E1 -1788.827,E2 -1788.827} C_VEL
LIN {X 0,Y 580.314,Z 399.202,A -85,B 0,C 180,E1 -1791.644,E2 -1791.644} C_VEL
LIN {X 0,Y 580.284,Z 399.206,A -85,B 0,C 180,E1 -1793.742,E2 -1793.742} C_VEL
LIN {X 0,Y 580.269,Z 399.208,A -85,B 0,C 180,E1 -1795.833,E2 -1795.833} C_VEL
LIN {X 0,Y 580.338,Z 399.2,A -85,B 0,C 180,E1 -1797.918,E2 -1797.918} C_VEL
LIN {X 0,Y 580.365,Z 399.194,A -85,B 0,C 180,E1 -1800.694,E2 -1800.694} C_VEL
LIN {X 0,Y 580.293,Z 399.203,A -85,B 0,C 180,E1 -1803.472,E2 -1803.472} C_VEL
LIN {X 0,Y 580.329,Z 399.199,A -85,B 0,C 180,E1 -1805.56,E2 -1805.56} C_VEL
LIN {X 0,Y 580.326,Z 399.2,A -85,B 0,C 180,E1 -1807.655,E2 -1807.655} C_VEL
LIN {X 0,Y 580.303,Z 399.204,A -85,B 0,C 180,E1 -1810.467,E2 -1810.467} C_VEL
LIN {X 0,Y 580.28,Z 399.204,A -85,B 0,C 180,E1 -1813.304,E2 -1813.304} C_VEL
LIN {X 0,Y 580.302,Z 399.202,A -85,B 0,C 180,E1 -1815.453,E2 -1815.453} C_VEL
LIN {X 0,Y 580.309,Z 399.201,A -85,B 0,C 180,E1 -1817.624,E2 -1817.624} C_VEL
LIN {X 0,Y 580.31,Z 399.201,A -85,B 0,C 180,E1 -1819.822,E2 -1819.822} C_VEL
LIN {X 0,Y 580.293,Z 399.203,A -85,B 0,C 180,E1 -1822.803,E2 -1822.803} C_VEL
LIN {X 0,Y 580.308,Z 399.201,A -85,B 0,C 180,E1 -1825.08,E2 -1825.08} C_VEL
LIN {X 0,Y 580.304,Z 399.202,A -85,B 0,C 180,E1 -1828.185,E2 -1828.185} C_VEL
LIN {X 0,Y 580.296,Z 399.205,A -85,B 0,C 180,E1 -1830.696,E2 -1830.696} C_VEL
LIN {X 0,Y 580.307,Z 399.201,A -85,B 0,C 180,E1 -1833.316,E2 -1833.316} C_VEL
LIN {X 0,Y 580.297,Z 399.202,A -85,B 0,C 180,E1 -1836.402,E2 -1836.402} C_VEL
LIN {X 0,Y 580.301,Z 399.204,A -85,B 0,C 180,E1 -1839.186,E2 -1839.186} C_VEL
LIN {X 0,Y 580.292,Z 399.203,A -85,B 0,C 180,E1 -1841.768,E2 -1841.768} C_VEL
LIN {X 0,Y 580.272,Z 399.207,A -85,B 0,C 180,E1 -1844.626,E2 -1844.626} C_VEL
LIN {X 0,Y 580.289,Z 399.206,A -85,B 0,C 180,E1 -1847.628,E2 -1847.628} C_VEL
LIN {X 0,Y 580.299,Z 399.203,A -85,B 0,C 180,E1 -1850.067,E2 -1850.067} C_VEL
LIN {X 0,Y 580.306,Z 399.204,A -85,B 0,C 180,E1 -1853.065,E2 -1853.065} C_VEL
LIN {X 0,Y 580.368,Z 399.296,A -85,B 0,C 180,E1 -1853.604,E2 -1853.604} C_VEL
LIN {X 0,Y 580.939,Z 404.583,A -85,B 0,C 180,E1 -1854.714,E2 -1854.714} C_VEL
LIN {X 0,Y 580.848,Z 420.699,A -85,B 0,C 180,E1 -1857.884,E2 -1857.884} C_VEL
LIN {X 0,Y 580.922,Z 434.891,A -85,B 0,C 180,E1 -1860.582,E2 -1860.582} C_VEL
LIN {X 0,Y 580.935,Z 445.799,A -85,B 0,C 180,E1 -1862.631,E2 -1862.631} C_VEL
LIN {X 0,Y 580.765,Z 460.08,A -85,B 0,C 180,E1 -1865.438,E2 -1865.438} C_VEL
LIN {X 0,Y 580.625,Z 473.189,A -85,B 0,C 180,E1 -1867.961,E2 -1867.961} C_VEL
LIN {X 0,Y 580.512,Z 488.14,A -85,B 0,C 180,E1 -1870.789,E2 -1870.789} C_VEL
LIN {X 0,Y 580.39,Z 502.535,A -85,B 0,C 180,E1 -1873.467,E2 -1873.467} C_VEL
LIN {X 0,Y 580.302,Z 518.187,A -85,B 0,C 180,E1 -1876.34,E2 -1876.34} C_VEL
LIN {X 0,Y 580.271,Z 525.156,A -85,B 0,C 180,E1 -1877.608,E2 -1877.608} C_VEL
LIN {X 0,Y 580.805,Z 530.946,A -85,B 0,C 180,E1 -1877.708,E2 -1877.708} C_VEL
LIN {X 0,Y 580.745,Z 544.219,A -85,B 0,C 180,E1 -1878.017,E2 -1878.017} C_VEL
LIN {X 0,Y 580.666,Z 556.372,A -85,B 0,C 180,E1 -1878.436,E2 -1878.436} C_VEL
LIN {X 0,Y 580.55,Z 568.631,A -85,B 0,C 180,E1 -1879.008,E2 -1879.008} C_VEL
LIN {X 0,Y 580.422,Z 580.202,A -85,B 0,C 180,E1 -1879.712,E2 -1879.712} C_VEL
LIN {X 0,Y 580.346,Z 590.598,A -85,B 0,C 180,E1 -1880.503,E2 -1880.503} C_VEL
LIN {X 0,Y 580.271,Z 599.112,A -85,B 0,C 180,E1 -1881.292,E2 -1881.292} C_VEL
LIN {X 0,Y 580.222,Z 606.961,A -85,B 0,C 180,E1 -1882.168,E2 -1882.168} C_VEL
LIN {X 0,Y 580.154,Z 614.65,A -85,B 0,C 180,E1 -1883.222,E2 -1883.222} C_VEL
LIN {X 0,Y 580.139,Z 621.68,A -85,B 0,C 180,E1 -1884.439,E2 -1884.439} C_VEL
LIN {X 0,Y 580.108,Z 626.372,A -85,B 0,C 180,E1 -1885.483,E2 -1885.483} C_VEL
LIN {X 0,Y 580.123,Z 629.957,A -85,B 0,C 180,E1 -1886.527,E2 -1886.527} C_VEL
LIN {X 0,Y 580.043,Z 631.809,A -85,B 0,C 180,E1 -1887.222,E2 -1887.222} C_VEL
LIN {X 0,Y 580.038,Z 633.2,A -85,B 0,C 180,E1 -1887.917,E2 -1887.917} C_VEL
LIN {X 0,Y 580.04,Z 634.784,A -85,B 0,C 180,E1 -1889.306,E2 -1889.306} C_VEL
LIN {X 0,Y 580.037,Z 635,A -85,B 0,C 180,E1 -1890,E2 -1890} C_VEL
LIN {X 0,Y 580.047,Z 634.185,A -85,B 0,C 180,E1 -1891.389,E2 -1891.389} C_VEL
LIN {X 0,Y 580.038,Z 633.201,A -85,B 0,C 180,E1 -1892.083,E2 -1892.083} C_VEL
LIN {X 0,Y 580.043,Z 631.81,A -85,B 0,C 180,E1 -1892.778,E2 -1892.778} C_VEL
LIN {X 0,Y 580.109,Z 628.896,A -85,B 0,C 180,E1 -1893.821,E2 -1893.821} C_VEL
LIN {X 0,Y 580.054,Z 624.949,A -85,B 0,C 180,E1 -1894.865,E2 -1894.865} C_VEL
LIN {X 0,Y 580.139,Z 618.877,A -85,B 0,C 180,E1 -1896.085,E2 -1896.085} C_VEL
LIN {X 0,Y 580.184,Z 612.236,A -85,B 0,C 180,E1 -1897.132,E2 -1897.132} C_VEL
LIN {X 0,Y 580.25,Z 603.989,A -85,B 0,C 180,E1 -1898.182,E2 -1898.182} C_VEL
LIN {X 0,Y 580.308,Z 595.537,A -85,B 0,C 180,E1 -1899.058,E2 -1899.058} C_VEL
LIN {X 0,Y 580.417,Z 585.094,A -85,B 0,C 180,E1 -1899.936,E2 -1899.936} C_VEL
LIN {X 0,Y 580.506,Z 574.755,A -85,B 0,C 180,E1 -1900.639,E2 -1900.639} C_VEL
LIN {X 0,Y 580.595,Z 563.259,A -85,B 0,C 180,E1 -1901.263,E2 -1901.263} C_VEL
LIN {X 0,Y 580.659,Z 550.468,A -85,B 0,C 180,E1 -1901.785,E2 -1901.785} C_VEL
LIN {X 0,Y 580.785,Z 537.43,A -85,B 0,C 180,E1 -1902.159,E2 -1902.159} C_VEL
LIN {X 0,Y 580.633,Z 527.535,A -85,B 0,C 180,E1 -1902.348,E2 -1902.348} C_VEL
LIN {X 0,Y 580.255,Z 525.034,A -85,B 0,C 180,E1 -1902.415,E2 -1902.415} C_VEL
LIN {X 0,Y 580.341,Z 510.36,A -85,B 0,C 180,E1 -1905.092,E2 -1905.092} C_VEL
LIN {X 0,Y 580.442,Z 494.709,A -85,B 0,C 180,E1 -1907.984,E2 -1907.984} C_VEL
LIN {X 0,Y 580.585,Z 479.221,A -85,B 0,C 180,E1 -1910.891,E2 -1910.891} C_VEL
LIN {X 0,Y 580.734,Z 463.406,A -85,B 0,C 180,E1 -1913.917,E2 -1913.917} C_VEL
LIN {X 0,Y 580.879,Z 449.711,A -85,B 0,C 180,E1 -1916.594,E2 -1916.594} C_VEL
LIN {X 0,Y 580.908,Z 439.544,A -85,B 0,C 180,E1 -1918.547,E2 -1918.547} C_VEL
LIN {X 0,Y 580.877,Z 426.38,A -85,B 0,C 180,E1 -1921.032,E2 -1921.032} C_VEL
LIN {X 0,Y 580.851,Z 411.942,A -85,B 0,C 180,E1 -1923.82,E2 -1923.82} C_VEL
LIN {X 0,Y 580.925,Z 403.534,A -85,B 0,C 180,E1 -1925.5,E2 -1925.5} C_VEL
LIN {X 0,Y 580.338,Z 399.199,A -85,B 0,C 180,E1 -1926.447,E2 -1926.447} C_VEL
LIN {X 0,Y 580.314,Z 399.202,A -85,B 0,C 180,E1 -1929.187,E2 -1929.187} C_VEL
LIN {X 0,Y 580.318,Z 399.199,A -85,B 0,C 180,E1 -1931.766,E2 -1931.766} C_VEL
LIN {X 0,Y 580.267,Z 399.208,A -85,B 0,C 180,E1 -1934.626,E2 -1934.626} C_VEL
LIN {X 0,Y 580.286,Z 399.204,A -85,B 0,C 180,E1 -1937.294,E2 -1937.294} C_VEL
LIN {X 0,Y 580.288,Z 399.204,A -85,B 0,C 180,E1 -1940.067,E2 -1940.067} C_VEL
LIN {X 0,Y 580.307,Z 399.203,A -85,B 0,C 180,E1 -1943.065,E2 -1943.065} C_VEL
LIN {X 0,Y 580.3,Z 399.202,A -85,B 0,C 180,E1 -1945.442,E2 -1945.442} C_VEL
LIN {X 0,Y 580.313,Z 399.201,A -85,B 0,C 180,E1 -1947.968,E2 -1947.968} C_VEL
LIN {X 0,Y 580.306,Z 399.201,A -85,B 0,C 180,E1 -1950.69,E2 -1950.69} C_VEL
LIN {X 0,Y 580.294,Z 399.205,A -85,B 0,C 180,E1 -1953.666,E2 -1953.666} C_VEL
LIN {X 0,Y 580.301,Z 399.204,A -85,B 0,C 180,E1 -1955.684,E2 -1955.684} C_VEL
LIN {X 0,Y 580.29,Z 399.205,A -85,B 0,C 180,E1 -1958.695,E2 -1958.695} C_VEL
LIN {X 0,Y 580.324,Z 399.201,A -85,B 0,C 180,E1 -1960.914,E2 -1960.914} C_VEL
LIN {X 0,Y 580.285,Z 399.204,A -85,B 0,C 180,E1 -1963.826,E2 -1963.826} C_VEL
LIN {X 0,Y 580.331,Z 399.199,A -85,B 0,C 180,E1 -1965.983,E2 -1965.983} C_VEL
LIN {X 0,Y 580.31,Z 399.201,A -85,B 0,C 180,E1 -1968.827,E2 -1968.827} C_VEL
LIN {X 0,Y 580.314,Z 399.203,A -85,B 0,C 180,E1 -1971.644,E2 -1971.644} C_VEL
LIN {X 0,Y 580.287,Z 399.206,A -85,B 0,C 180,E1 -1973.742,E2 -1973.742} C_VEL
LIN {X 0,Y 580.276,Z 399.208,A -85,B 0,C 180,E1 -1975.833,E2 -1975.833} C_VEL
LIN {X 0,Y 580.345,Z 399.199,A -85,B 0,C 180,E1 -1977.918,E2 -1977.918} C_VEL
LIN {X 0,Y 580.369,Z 399.193,A -85,B 0,C 180,E1 -1980.694,E2 -1980.694} C_VEL
LIN {X 0,Y 580.29,Z 399.204,A -85,B 0,C 180,E1 -1983.472,E2 -1983.472} C_VEL
LIN {X 0,Y 580.325,Z 399.2,A -85,B 0,C 180,E1 -1985.56,E2 -1985.56} C_VEL
LIN {X 0,Y 580.327,Z 399.2,A -85,B 0,C 180,E1 -1987.655,E2 -1987.655} C_VEL
LIN {X 0,Y 580.306,Z 399.202,A -85,B 0,C 180,E1 -1990.467,E2 -1990.467} C_VEL
LIN {X 0,Y 580.279,Z 399.205,A -85,B 0,C 180,E1 -1993.304,E2 -1993.304} C_VEL
LIN {X 0,Y 580.302,Z 399.202,A -85,B 0,C 180,E1 -1995.453,E2 -1995.453} C_VEL
LIN {X 0,Y 580.299,Z 399.202,A -85,B 0,C 180,E1 -1997.624,E2 -1997.624} C_VEL
LIN {X 0,Y 580.31,Z 399.201,A -85,B 0,C 180,E1 -1999.822,E2 -1999.822} C_VEL
LIN {X 0,Y 580.288,Z 399.206,A -85,B 0,C 180,E1 -2001.331,E2 -2001.331} C_VEL
LIN {X 0,Y 579.59,Z 399.291,A -85,B 0,C 180,E1 -2001.91,E2 -2001.91} C_VEL
LIN {X 0,Y 576.71,Z 399.649,A -85,B 0,C 180,E1 -2002.85,E2 -2002.85} C_VEL
LIN {X 0,Y 574.315,Z 399.948,A -85,B 0,C 180,E1 -2003.606,E2 -2003.606} C_VEL
LIN {X 0,Y 573.317,Z 400.072,A -85,B 0,C 180,E1 -2004.19,E2 -2004.19} C_VEL
LIN {X 0,Y 573.252,Z 400.079,A -85,B 0,C 180,E1 -2004.387,E2 -2004.387} C_VEL
LIN {X 0,Y 573.256,Z 400.08,A -85,B 0,C 180,E1 -2006.976,E2 -2006.976} C_VEL
LIN {X 0,Y 573.253,Z 400.081,A -85,B 0,C 180,E1 -2009.489,E2 -2009.489} C_VEL
LIN {X 0,Y 573.261,Z 400.079,A -85,B 0,C 180,E1 -2012.229,E2 -2012.229} C_VEL
LIN {X 0,Y 573.24,Z 400.082,A -85,B 0,C 180,E1 -2014.771,E2 -2014.771} C_VEL
LIN {X 0,Y 573.238,Z 400.082,A -85,B 0,C 180,E1 -2017.808,E2 -2017.808} C_VEL
LIN {X 0,Y 573.248,Z 400.082,A -85,B 0,C 180,E1 -2020.525,E2 -2020.525} C_VEL
LIN {X 0,Y 573.251,Z 400.082,A -85,B 0,C 180,E1 -2023.358,E2 -2023.358} C_VEL
LIN {X 0,Y 573.257,Z 400.079,A -85,B 0,C 180,E1 -2026.33,E2 -2026.33} C_VEL
LIN {X 0,Y 573.279,Z 400.077,A -85,B 0,C 180,E1 -2029.477,E2 -2029.477} C_VEL
LIN {X 0,Y 573.24,Z 400.083,A -85,B 0,C 180,E1 -2032.193,E2 -2032.193} C_VEL
LIN {X 0,Y 573.242,Z 400.083,A -85,B 0,C 180,E1 -2035.228,E2 -2035.228} C_VEL
LIN {X 0,Y 573.255,Z 400.079,A -85,B 0,C 180,E1 -2037.772,E2 -2037.772} C_VEL
LIN {X 0,Y 573.271,Z 400.079,A -85,B 0,C 180,E1 -2040.634,E2 -2040.634} C_VEL
LIN {X 0,Y 573.243,Z 400.083,A -85,B 0,C 180,E1 -2043.507,E2 -2043.507} C_VEL
LIN {X 0,Y 573.237,Z 400.082,A -85,B 0,C 180,E1 -2046.135,E2 -2046.135} C_VEL
LIN {X 0,Y 573.254,Z 400.08,A -85,B 0,C 180,E1 -2049.174,E2 -2049.174} C_VEL
LIN {X 0,Y 573.224,Z 400.083,A -85,B 0,C 180,E1 -2051.411,E2 -2051.411} C_VEL
LIN {X 0,Y 573.252,Z 400.08,A -85,B 0,C 180,E1 -2053.622,E2 -2053.622} C_VEL
LIN {X 0,Y 573.278,Z 400.077,A -85,B 0,C 180,E1 -2055.807,E2 -2055.807} C_VEL
LIN {X 0,Y 573.278,Z 400.077,A -85,B 0,C 180,E1 -2058.083,E2 -2058.083} C_VEL
LIN {X 0,Y 573.729,Z 404.145,A -85,B 0,C 180,E1 -2058.25,E2 -2058.25} C_VEL
LIN {X 0,Y 573.6,Z 416.763,A -85,B 0,C 180,E1 -2058.821,E2 -2058.821} C_VEL
LIN {X 0,Y 573.479,Z 428.262,A -85,B 0,C 180,E1 -2059.497,E2 -2059.497} C_VEL
LIN {X 0,Y 573.351,Z 439.001,A -85,B 0,C 180,E1 -2060.297,E2 -2060.297} C_VEL
LIN {X 0,Y 573.241,Z 448.67,A -85,B 0,C 180,E1 -2061.185,E2 -2061.185} C_VEL
LIN {X 0,Y 573.161,Z 456.596,A -85,B 0,C 180,E1 -2062.071,E2 -2062.071} C_VEL
LIN {X 0,Y 573.089,Z 464.565,A -85,B 0,C 180,E1 -2063.168,E2 -2063.168} C_VEL
LIN {X 0,Y 573.071,Z 471.463,A -85,B 0,C 180,E1 -2064.37,E2 -2064.37} C_VEL
LIN {X 0,Y 573.029,Z 476.202,A -85,B 0,C 180,E1 -2065.427,E2 -2065.427} C_VEL
LIN {X 0,Y 573.022,Z 479.832,A -85,B 0,C 180,E1 -2066.484,E2 -2066.484} C_VEL
LIN {X 0,Y 572.959,Z 481.693,A -85,B 0,C 180,E1 -2067.188,E2 -2067.188} C_VEL
LIN {X 0,Y 572.939,Z 483.135,A -85,B 0,C 180,E1 -2067.891,E2 -2067.891} C_VEL
LIN {X 0,Y 572.941,Z 484.755,A -85,B 0,C 180,E1 -2069.297,E2 -2069.297} C_VEL
LIN {X 0,Y 572.939,Z 484.996,A -85,B 0,C 180,E1 -2070,E2 -2070} C_VEL
LIN {X 0,Y 572.94,Z 484.813,A -85,B 0,C 180,E1 -2070.703,E2 -2070.703} C_VEL
LIN {X 0,Y 572.94,Z 483.275,A -85,B 0,C 180,E1 -2072.109,E2 -2072.109} C_VEL
LIN {X 0,Y 572.96,Z 481.908,A -85,B 0,C 180,E1 -2072.812,E2 -2072.812} C_VEL
LIN {X 0,Y 573.015,Z 479.039,A -85,B 0,C 180,E1 -2073.868,E2 -2073.868} C_VEL
LIN {X 0,Y 572.963,Z 475.14,A -85,B 0,C 180,E1 -2074.926,E2 -2074.926} C_VEL
LIN {X 0,Y 573.075,Z 470.097,A -85,B 0,C 180,E1 -2075.983,E2 -2075.983} C_VEL
LIN {X 0,Y 573.083,Z 463.765,A -85,B 0,C 180,E1 -2077.044,E2 -2077.044} C_VEL
LIN {X 0,Y 573.175,Z 455.867,A -85,B 0,C 180,E1 -2078.106,E2 -2078.106} C_VEL
LIN {X 0,Y 573.254,Z 447.795,A -85,B 0,C 180,E1 -2078.993,E2 -2078.993} C_VEL
LIN {X 0,Y 573.346,Z 437.945,A -85,B 0,C 180,E1 -2079.881,E2 -2079.881} C_VEL
LIN {X 0,Y 573.529,Z 426.933,A -85,B 0,C 180,E1 -2080.678,E2 -2080.678} C_VEL
LIN {X 0,Y 573.58,Z 416.071,A -85,B 0,C 180,E1 -2081.306,E2 -2081.306} C_VEL
LIN {X 0,Y 573.716,Z 404.16,A -85,B 0,C 180,E1 -2081.84,E2 -2081.84} C_VEL
LIN {X 0,Y 573.355,Z 400.519,A -85,B 0,C 180,E1 -2081.983,E2 -2081.983} C_VEL
LIN {X 0,Y 573.294,Z 400.075,A -85,B 0,C 180,E1 -2082.029,E2 -2082.029} C_VEL
LIN {X 0,Y 573.239,Z 400.083,A -85,B 0,C 180,E1 -2084.92,E2 -2084.92} C_VEL
LIN {X 0,Y 573.246,Z 400.083,A -85,B 0,C 180,E1 -2087.848,E2 -2087.848} C_VEL
LIN {X 0,Y 573.246,Z 400.084,A -85,B 0,C 180,E1 -2090.077,E2 -2090.077} C_VEL
LIN {X 0,Y 573.242,Z 400.083,A -85,B 0,C 180,E1 -2092.338,E2 -2092.338} C_VEL
LIN {X 0,Y 573.26,Z 400.081,A -85,B 0,C 180,E1 -2095.41,E2 -2095.41} C_VEL
LIN {X 0,Y 573.269,Z 400.077,A -85,B 0,C 180,E1 -2098.031,E2 -2098.031} C_VEL
LIN {X 0,Y 573.233,Z 400.084,A -85,B 0,C 180,E1 -2100.882,E2 -2100.882} C_VEL
LIN {X 0,Y 573.266,Z 400.079,A -85,B 0,C 180,E1 -2103.524,E2 -2103.524} C_VEL
LIN {X 0,Y 573.263,Z 400.08,A -85,B 0,C 180,E1 -2106.048,E2 -2106.048} C_VEL
LIN {X 0,Y 573.254,Z 400.08,A -85,B 0,C 180,E1 -2108.701,E2 -2108.701} C_VEL
LIN {X 0,Y 573.257,Z 400.079,A -85,B 0,C 180,E1 -2111.596,E2 -2111.596} C_VEL
LIN {X 0,Y 573.243,Z 400.082,A -85,B 0,C 180,E1 -2114.333,E2 -2114.333} C_VEL
LIN {X 0,Y 573.247,Z 400.082,A -85,B 0,C 180,E1 -2117.358,E2 -2117.358} C_VEL
LIN {X 0,Y 573.242,Z 400.081,A -85,B 0,C 180,E1 -2120.392,E2 -2120.392} C_VEL
LIN {X 0,Y 573.256,Z 400.081,A -85,B 0,C 180,E1 -2123.078,E2 -2123.078} C_VEL
LIN {X 0,Y 573.272,Z 400.077,A -85,B 0,C 180,E1 -2125.671,E2 -2125.671} C_VEL
LIN {X 0,Y 573.249,Z 400.082,A -85,B 0,C 180,E1 -2128.185,E2 -2128.185} C_VEL
LIN {X 0,Y 573.269,Z 400.078,A -85,B 0,C 180,E1 -2130.634,E2 -2130.634} C_VEL
LIN {X 0,Y 573.254,Z 400.08,A -85,B 0,C 180,E1 -2133.024,E2 -2133.024} C_VEL
LIN {X 0,Y 573.277,Z 400.078,A -85,B 0,C 180,E1 -2135.366,E2 -2135.366} C_VEL
LIN {X 0,Y 573.233,Z 400.083,A -85,B 0,C 180,E1 -2138.419,E2 -2138.419} C_VEL
LIN {X 0,Y 573.282,Z 400.078,A -85,B 0,C 180,E1 -2140.728,E2 -2140.728} C_VEL
LIN {X 0,Y 573.257,Z 400.079,A -85,B 0,C 180,E1 -2143.622,E2 -2143.622} C_VEL
LIN {X 0,Y 573.278,Z 400.076,A -85,B 0,C 180,E1 -2145.807,E2 -2145.807} C_VEL
LIN {X 0,Y 573.267,Z 400.078,A -85,B 0,C 180,E1 -2148.745,E2 -2148.745} C_VEL
LIN {X 0,Y 573.258,Z 400.081,A -85,B 0,C 180,E1 -2151.54,E2 -2151.54} C_VEL
LIN {X 0,Y 573.246,Z 400.083,A -85,B 0,C 180,E1 -2153.665,E2 -2153.665} C_VEL
LIN {X 0,Y 573.227,Z 400.085,A -85,B 0,C 180,E1 -2155.781,E2 -2155.781} C_VEL
LIN {X 0,Y 573.31,Z 400.075,A -85,B 0,C 180,E1 -2157.892,E2 -2157.892} C_VEL
LIN {X 0,Y 573.336,Z 400.07,A -85,B 0,C 180,E1 -2160.702,E2 -2160.702} C_VEL
LIN {X 0,Y 573.245,Z 400.081,A -85,B 0,C 180,E1 -2163.514,E2 -2163.514} C_VEL
LIN {X 0,Y 573.296,Z 400.075,A -85,B 0,C 180,E1 -2165.628,E2 -2165.628} C_VEL
LIN {X 0,Y 573.274,Z 400.077,A -85,B 0,C 180,E1 -2167.75,E2 -2167.75} C_VEL
LIN {X 0,Y 573.27,Z 400.08,A -85,B 0,C 180,E1 -2170.597,E2 -2170.597} C_VEL
LIN {X 0,Y 573.27,Z 400.079,A -85,B 0,C 180,E1 -2172.748,E2 -2172.748} C_VEL
LIN {X 0,Y 573.241,Z 400.082,A -85,B 0,C 180,E1 -2174.92,E2 -2174.92} C_VEL
LIN {X 0,Y 573.259,Z 400.081,A -85,B 0,C 180,E1 -2177.848,E2 -2177.848} C_VEL
LIN {X 0,Y 573.257,Z 400.082,A -85,B 0,C 180,E1 -2180.077,E2 -2180.077} C_VEL
LIN {X 0,Y 573.238,Z 400.083,A -85,B 0,C 180,E1 -2183.099,E2 -2183.099} C_VEL
LIN {X 0,Y 573.256,Z 400.082,A -85,B 0,C 180,E1 -2185.41,E2 -2185.41} C_VEL
LIN {X 0,Y 573.256,Z 400.08,A -85,B 0,C 180,E1 -2188.029,E2 -2188.029} C_VEL
LIN {X 0,Y 573.242,Z 400.082,A -85,B 0,C 180,E1 -2190.884,E2 -2190.884} C_VEL
LIN {X 0,Y 573.265,Z 400.078,A -85,B 0,C 180,E1 -2193.524,E2 -2193.524} C_VEL
LIN {X 0,Y 573.261,Z 400.081,A -85,B 0,C 180,E1 -2196.048,E2 -2196.048} C_VEL
LIN {X 0,Y 573.246,Z 400.08,A -85,B 0,C 180,E1 -2198.701,E2 -2198.701} C_VEL
LIN {X 0,Y 573.239,Z 400.082,A -85,B 0,C 180,E1 -2201.594,E2 -2201.594} C_VEL
LIN {X 0,Y 573.243,Z 400.083,A -85,B 0,C 180,E1 -2204.333,E2 -2204.333} C_VEL
LIN {X 0,Y 573.244,Z 400.082,A -85,B 0,C 180,E1 -2207.358,E2 -2207.358} C_VEL
LIN {X 0,Y 573.252,Z 400.08,A -85,B 0,C 180,E1 -2210.393,E2 -2210.393} C_VEL
LIN {X 0,Y 573.297,Z 400.181,A -85,B 0,C 180,E1 -2213.41,E2 -2213.41} C_VEL
LIN {X 0,Y 573.981,Z 404.909,A -85,B 0,C 180,E1 -2214.436,E2 -2214.436} C_VEL
LIN {X 0,Y 573.901,Z 419.711,A -85,B 0,C 180,E1 -2217.396,E2 -2217.396} C_VEL
LIN {X 0,Y 573.925,Z 434.057,A -85,B 0,C 180,E1 -2220.168,E2 -2220.168} C_VEL
LIN {X 0,Y 573.919,Z 449.46,A -85,B 0,C 180,E1 -2223.058,E2 -2223.058} C_VEL
LIN {X 0,Y 573.821,Z 461.45,A -85,B 0,C 180,E1 -2225.391,E2 -2225.391} C_VEL
LIN {X 0,Y 573.637,Z 475.145,A -85,B 0,C 180,E1 -2228.057,E2 -2228.057} C_VEL
LIN {X 0,Y 573.502,Z 488.84,A -85,B 0,C 180,E1 -2230.678,E2 -2230.678} C_VEL
LIN {X 0,Y 573.362,Z 502.687,A -85,B 0,C 180,E1 -2233.287,E2 -2233.287} C_VEL
LIN {X 0,Y 573.252,Z 518.187,A -85,B 0,C 180,E1 -2236.168,E2 -2236.168} C_VEL
LIN {X 0,Y 573.191,Z 525.156,A -85,B 0,C 180,E1 -2237.452,E2 -2237.452} C_VEL
LIN {X 0,Y 573.863,Z 530.946,A -85,B 0,C 180,E1 -2237.557,E2 -2237.557} C_VEL
LIN {X 0,Y 573.81,Z 544.219,A -85,B 0,C 180,E1 -2237.87,E2 -2237.87} C_VEL
LIN {X 0,Y 573.714,Z 556.373,A -85,B 0,C 180,E1 -2238.294,E2 -2238.294} C_VEL
LIN {X 0,Y 573.586,Z 568.66,A -85,B 0,C 180,E1 -2238.875,E2 -2238.875} C_VEL
LIN {X 0,Y 573.434,Z 580.203,A -85,B 0,C 180,E1 -2239.585,E2 -2239.585} C_VEL
LIN {X 0,Y 573.334,Z 590.599,A -85,B 0,C 180,E1 -2240.386,E2 -2240.386} C_VEL
LIN {X 0,Y 573.241,Z 599.113,A -85,B 0,C 180,E1 -2241.185,E2 -2241.185} C_VEL
LIN {X 0,Y 573.161,Z 606.961,A -85,B 0,C 180,E1 -2242.071,E2 -2242.071} C_VEL
LIN {X 0,Y 573.072,Z 614.954,A -85,B 0,C 180,E1 -2243.185,E2 -2243.185} C_VEL
LIN {X 0,Y 573.07,Z 621.68,A -85,B 0,C 180,E1 -2244.37,E2 -2244.37} C_VEL
LIN {X 0,Y 573.029,Z 626.372,A -85,B 0,C 180,E1 -2245.428,E2 -2245.428} C_VEL
LIN {X 0,Y 573.022,Z 629.957,A -85,B 0,C 180,E1 -2246.484,E2 -2246.484} C_VEL
LIN {X 0,Y 572.959,Z 631.808,A -85,B 0,C 180,E1 -2247.188,E2 -2247.188} C_VEL
LIN {X 0,Y 572.938,Z 633.199,A -85,B 0,C 180,E1 -2247.891,E2 -2247.891} C_VEL
LIN {X 0,Y 572.94,Z 634.785,A -85,B 0,C 180,E1 -2249.297,E2 -2249.297} C_VEL
LIN {X 0,Y 572.938,Z 635,A -85,B 0,C 180,E1 -2250,E2 -2250} C_VEL
LIN {X 0,Y 572.946,Z 634.186,A -85,B 0,C 180,E1 -2251.406,E2 -2251.406} C_VEL
LIN {X 0,Y 572.938,Z 633.2,A -85,B 0,C 180,E1 -2252.109,E2 -2252.109} C_VEL
LIN {X 0,Y 572.959,Z 631.81,A -85,B 0,C 180,E1 -2252.812,E2 -2252.812} C_VEL
LIN {X 0,Y 573.014,Z 628.896,A -85,B 0,C 180,E1 -2253.868,E2 -2253.868} C_VEL
LIN {X 0,Y 572.963,Z 624.949,A -85,B 0,C 180,E1 -2254.926,E2 -2254.926} C_VEL
LIN {X 0,Y 573.064,Z 618.876,A -85,B 0,C 180,E1 -2256.16,E2 -2256.16} C_VEL
LIN {X 0,Y 573.119,Z 612.237,A -85,B 0,C 180,E1 -2257.221,E2 -2257.221} C_VEL
LIN {X 0,Y 573.201,Z 603.989,A -85,B 0,C 180,E1 -2258.283,E2 -2258.283} C_VEL
LIN {X 0,Y 573.287,Z 595.537,A -85,B 0,C 180,E1 -2259.17,E2 -2259.17} C_VEL
LIN {X 0,Y 573.421,Z 585.095,A -85,B 0,C 180,E1 -2260.059,E2 -2260.059} C_VEL
LIN {X 0,Y 573.548,Z 573.437,A -85,B 0,C 180,E1 -2260.853,E2 -2260.853} C_VEL
LIN {X 0,Y 573.65,Z 562.314,A -85,B 0,C 180,E1 -2261.446,E2 -2261.446} C_VEL
LIN {X 0,Y 573.731,Z 549.17,A -85,B 0,C 180,E1 -2261.975,E2 -2261.975} C_VEL
LIN {X 0,Y 573.854,Z 536.515,A -85,B 0,C 180,E1 -2262.331,E2 -2262.331} C_VEL
LIN {X 0,Y 573.611,Z 527.722,A -85,B 0,C 180,E1 -2262.499,E2 -2262.499} C_VEL
LIN {X 0,Y 573.194,Z 525.034,A -85,B 0,C 180,E1 -2262.57,E2 -2262.57} C_VEL
LIN {X 0,Y 573.316,Z 510.36,A -85,B 0,C 180,E1 -2265.281,E2 -2265.281} C_VEL
LIN {X 0,Y 573.461,Z 494.709,A -85,B 0,C 180,E1 -2268.211,E2 -2268.211} C_VEL
LIN {X 0,Y 573.598,Z 479.54,A -85,B 0,C 180,E1 -2271.096,E2 -2271.096} C_VEL
LIN {X 0,Y 573.776,Z 465.362,A -85,B 0,C 180,E1 -2273.842,E2 -2273.842} C_VEL
LIN {X 0,Y 573.937,Z 451.132,A -85,B 0,C 180,E1 -2276.632,E2 -2276.632} C_VEL
LIN {X 0,Y 573.92,Z 436.695,A -85,B 0,C 180,E1 -2279.329,E2 -2279.329} C_VEL
LIN {X 0,Y 573.908,Z 422.541,A -85,B 0,C 180,E1 -2282.05,E2 -2282.05} C_VEL
LIN {X 0,Y 574.005,Z 405.975,A -85,B 0,C 180,E1 -2285.347,E2 -2285.347} C_VEL
LIN {X 0,Y 573.405,Z 400.693,A -85,B 0,C 180,E1 -2286.473,E2 -2286.473} C_VEL
LIN {X 0,Y 573.304,Z 400.076,A -85,B 0,C 180,E1 -2286.645,E2 -2286.645} C_VEL
LIN {X 0,Y 573.253,Z 400.081,A -85,B 0,C 180,E1 -2289.607,E2 -2289.607} C_VEL
LIN {X 0,Y 573.245,Z 400.082,A -85,B 0,C 180,E1 -2292.642,E2 -2292.642} C_VEL
LIN {X 0,Y 573.244,Z 400.083,A -85,B 0,C 180,E1 -2295.667,E2 -2295.667} C_VEL
LIN {X 0,Y 573.247,Z 400.082,A -85,B 0,C 180,E1 -2298.544,E2 -2298.544} C_VEL
LIN {X 0,Y 573.247,Z 400.08,A -85,B 0,C 180,E1 -2301.299,E2 -2301.299} C_VEL
LIN {X 0,Y 573.264,Z 400.081,A -85,B 0,C 180,E1 -2304.012,E2 -2304.012} C_VEL
LIN {X 0,Y 573.273,Z 400.077,A -85,B 0,C 180,E1 -2306.518,E2 -2306.518} C_VEL
LIN {X 0,Y 573.243,Z 400.082,A -85,B 0,C 180,E1 -2309.116,E2 -2309.116} C_VEL
LIN {X 0,Y 573.256,Z 400.08,A -85,B 0,C 180,E1 -2311.971,E2 -2311.971} C_VEL
LIN {X 0,Y 573.256,Z 400.082,A -85,B 0,C 180,E1 -2314.59,E2 -2314.59} C_VEL
LIN {X 0,Y 573.24,Z 400.083,A -85,B 0,C 180,E1 -2317.662,E2 -2317.662} C_VEL
LIN {X 0,Y 573.283,Z 400.077,A -85,B 0,C 180,E1 -2320.728,E2 -2320.728} C_VEL
LIN {X 0,Y 573.257,Z 400.079,A -85,B 0,C 180,E1 -2323.622,E2 -2323.622} C_VEL
LIN {X 0,Y 573.278,Z 400.077,A -85,B 0,C 180,E1 -2325.807,E2 -2325.807} C_VEL
LIN {X 0,Y 573.268,Z 400.078,A -85,B 0,C 180,E1 -2328.745,E2 -2328.745} C_VEL
LIN {X 0,Y 573.258,Z 400.081,A -85,B 0,C 180,E1 -2331.54,E2 -2331.54} C_VEL
LIN {X 0,Y 573.249,Z 400.083,A -85,B 0,C 180,E1 -2333.665,E2 -2333.665} C_VEL
LIN {X 0,Y 573.234,Z 400.085,A -85,B 0,C 180,E1 -2335.781,E2 -2335.781} C_VEL
LIN {X 0,Y 573.316,Z 400.075,A -85,B 0,C 180,E1 -2337.892,E2 -2337.892} C_VEL
LIN {X 0,Y 573.339,Z 400.068,A -85,B 0,C 180,E1 -2340.702,E2 -2340.702} C_VEL
LIN {X 0,Y 573.241,Z 400.082,A -85,B 0,C 180,E1 -2343.515,E2 -2343.515} C_VEL
LIN {X 0,Y 573.292,Z 400.076,A -85,B 0,C 180,E1 -2345.628,E2 -2345.628} C_VEL
LIN {X 0,Y 573.275,Z 400.078,A -85,B 0,C 180,E1 -2347.75,E2 -2347.75} C_VEL
LIN {X 0,Y 573.272,Z 400.079,A -85,B 0,C 180,E1 -2350.597,E2 -2350.597} C_VEL
LIN {X 0,Y 573.27,Z 400.079,A -85,B 0,C 180,E1 -2352.749,E2 -2352.749} C_VEL
LIN {X 0,Y 573.242,Z 400.083,A -85,B 0,C 180,E1 -2354.92,E2 -2354.92} C_VEL
LIN {X 0,Y 573.25,Z 400.081,A -85,B 0,C 180,E1 -2357.848,E2 -2357.848} C_VEL
LIN {X 0,Y 573.257,Z 400.081,A -85,B 0,C 180,E1 -2360.077,E2 -2360.077} C_VEL
